    movel([0.119613, -1.324282, -2.607686, -0.780421, 1.570796, 1.690410],accel_mss,speed_ms,0,blend_radius_m)
    movel([0.119842, -1.324467, -2.607569, -0.780352, 1.570796, 1.690638],accel_mss,speed_ms,0,blend_radius_m)
    movel([0.121399, -1.324125, -2.607784, -0.780480, 1.570796, 1.692195],accel_mss,speed_ms,0,blend_radius_m)
    movel([0.123082, -1.323676, -2.608066, -0.780647, 1.570796, 1.693878],accel_mss,speed_ms,0,blend_radius_m)
    movel([0.126728, -1.322614, -2.608731, -0.781044, 1.570796, 1.697525],accel_mss,speed_ms,0,blend_radius_m)
    movel([0.135559, -1.320026, -2.610347, -0.782016, 1.570796, 1.706355],accel_mss,speed_ms,0,blend_radius_m)
    movel([0.136875, -1.312057, -2.615265, -0.785067, 1.570796, 1.707671],accel_mss,speed_ms,0,blend_radius_m)
    movel([0.137268, -1.309610, -2.616758, -0.786021, 1.570796, 1.708065],accel_mss,speed_ms,0,blend_radius_m)
    movel([0.137372, -1.308887, -2.617198, -0.786304, 1.570796, 1.708168],accel_mss,speed_ms,0,blend_radius_m)
    movel([0.137487, -1.307784, -2.617868, -0.786738, 1.570796, 1.708283],accel_mss,speed_ms,0,blend_radius_m)
    movel([0.137501, -1.307407, -2.618096, -0.786886, 1.570796, 1.708297],accel_mss,speed_ms,0,blend_radius_m)
    movel([0.137496, -1.307037, -2.618320, -0.787032, 1.570796, 1.708292],accel_mss,speed_ms,0,blend_radius_m)
    movel([0.137349, -1.306827, -2.618447, -0.787115, 1.570796, 1.708145],accel_mss,speed_ms,0,blend_radius_m)
    movel([0.137251, -1.309745, -2.619823, -0.782821, 1.570796, 1.708047],accel_mss,speed_ms,0,blend_radius_m)
    movel([0.136956, -1.309738, -2.619827, -0.782824, 1.570796, 1.707752],accel_mss,speed_ms,0,blend_radius_m)
    movel([0.136646, -1.309759, -2.619814, -0.782816, 1.570796, 1.707442],accel_mss,speed_ms,0,blend_radius_m)
    movel([0.136330, -1.309805, -2.619786, -0.782797, 1.570796, 1.707126],accel_mss,speed_ms,0,blend_radius_m)
    movel([0.136004, -1.309880, -2.619741, -0.782768, 1.570796, 1.706800],accel_mss,speed_ms,0,blend_radius_m)
    movel([0.130263, -1.311569, -2.618712, -0.782108, 1.570796, 1.701060],accel_mss,speed_ms,0,blend_radius_m)
    movel([0.122240, -1.314022, -2.617212, -0.781155, 1.570796, 1.693036],accel_mss,speed_ms,0,blend_radius_m)
    movel([0.121881, -1.314196, -2.617105, -0.781088, 1.570796, 1.692677],accel_mss,speed_ms,0,blend_radius_m)
    movel([0.121557, -1.314459, -2.616944, -0.780986, 1.570796, 1.692353],accel_mss,speed_ms,0,blend_radius_m)
    movel([0.121274, -1.314831, -2.616715, -0.780843, 1.570796, 1.692071],accel_mss,speed_ms,0,blend_radius_m)
    movel([0.121125, -1.315219, -2.616477, -0.780693, 1.570796, 1.691922],accel_mss,speed_ms,0,blend_radius_m)
    movel([0.120597, -1.318726, -2.614312, -0.779350, 1.570796, 1.691393],accel_mss,speed_ms,0,blend_radius_m)
    movel([0.120081, -1.322273, -2.612107, -0.778009, 1.570796, 1.690877],accel_mss,speed_ms,0,blend_radius_m)
    movel([0.119488, -1.326560, -2.609418, -0.776411, 1.570796, 1.690285],accel_mss,speed_ms,0,blend_radius_m)
    movel([0.119491, -1.326786, -2.609276, -0.776327, 1.570796, 1.690287],accel_mss,speed_ms,0,blend_radius_m)
    movel([0.119613, -1.327186, -2.609024, -0.776179, 1.570796, 1.690410],accel_mss,speed_ms,0,blend_radius_m)
    movel([0.119842, -1.327371, -2.608907, -0.776111, 1.570796, 1.690638],accel_mss,speed_ms,0,blend_radius_m)
    movel([0.121399, -1.327030, -2.609122, -0.776237, 1.570796, 1.692195],accel_mss,speed_ms,0,blend_radius_m)
    movel([0.123082, -1.326582, -2.609405, -0.776403, 1.570796, 1.693878],accel_mss,speed_ms,0,blend_radius_m)
    movel([0.126728, -1.325522, -2.610072, -0.776796, 1.570796, 1.697525],accel_mss,speed_ms,0,blend_radius_m)
    movel([0.135559, -1.322939, -2.611691, -0.777759, 1.570796, 1.706355],accel_mss,speed_ms,0,blend_radius_m)
    movel([0.136875, -1.314985, -2.616621, -0.780783, 1.570796, 1.707671],accel_mss,speed_ms,0,blend_radius_m)
    movel([0.137268, -1.312544, -2.618117, -0.781728, 1.570796, 1.708065],accel_mss,speed_ms,0,blend_radius_m)
    movel([0.137372, -1.311822, -2.618558, -0.782009, 1.570796, 1.708168],accel_mss,speed_ms,0,blend_radius_m)
    movel([0.137487, -1.310721, -2.619229, -0.782439, 1.570796, 1.708283],accel_mss,speed_ms,0,blend_radius_m)
    movel([0.137501, -1.310344, -2.619458, -0.782586, 1.570796, 1.708297],accel_mss,speed_ms,0,blend_radius_m)
    movel([0.137496, -1.309975, -2.619683, -0.782731, 1.570796, 1.708292],accel_mss,speed_ms,0,blend_radius_m)
    movel([0.137349, -1.309765, -2.619810, -0.782813, 1.570796, 1.708145],accel_mss,speed_ms,0,blend_radius_m)
    movel([0.137251, -1.275756, -2.603080, -0.833553, 1.570796, 1.708047],accel_mss,speed_ms,0,blend_radius_m)
    speed_ms = 1.000
    movel([0.134220, -1.265196, -2.609125, -0.838068, 1.570796, 1.705016],accel_mss,speed_ms,0,blend_radius_m)
    speed_ms = 0.008
    movel([0.134220, -1.292915, -2.623010, -0.796463, 1.570796, 1.705016],accel_mss,speed_ms,0,blend_radius_m)
    speed_ms = 0.003
    movel([0.134220, -1.296430, -2.624667, -0.791291, 1.570796, 1.705016],accel_mss,speed_ms,0,blend_radius_m)
    speed_ms = 0.008
    movel([0.121435, -1.300332, -2.622350, -0.789708, 1.570796, 1.692232],accel_mss,speed_ms,0,blend_radius_m)
    movel([0.125336, -1.272015, -2.638732, -0.801642, 1.570796, 1.696133],accel_mss,speed_ms,0,blend_radius_m)
    movel([0.151954, -1.263834, -2.643278, -0.805277, 1.570796, 1.722750],accel_mss,speed_ms,0,blend_radius_m)
    movel([0.147041, -1.292633, -2.626904, -0.792852, 1.570796, 1.717838],accel_mss,speed_ms,0,blend_radius_m)
    movel([0.134220, -1.296430, -2.624667, -0.791291, 1.570796, 1.705016],accel_mss,speed_ms,0,blend_radius_m)
    movel([0.134220, -1.299389, -2.626045, -0.786955, 1.570796, 1.705016],accel_mss,speed_ms,0,blend_radius_m)
    movel([0.121435, -1.303283, -2.623722, -0.785384, 1.570796, 1.692232],accel_mss,speed_ms,0,blend_radius_m)
    movel([0.125336, -1.275018, -2.640145, -0.797226, 1.570796, 1.696133],accel_mss,speed_ms,0,blend_radius_m)
    movel([0.151954, -1.266851, -2.644703, -0.800836, 1.570796, 1.722750],accel_mss,speed_ms,0,blend_radius_m)
    movel([0.147041, -1.295599, -2.628288, -0.788502, 1.570796, 1.717838],accel_mss,speed_ms,0,blend_radius_m)
    movel([0.134220, -1.299389, -2.626045, -0.786955, 1.570796, 1.705016],accel_mss,speed_ms,0,blend_radius_m)
    movel([0.134220, -1.265196, -2.609125, -0.838068, 1.570796, 1.705016],accel_mss,speed_ms,0,blend_radius_m)
    speed_ms = 1.000
    movel([0.114823, -1.278281, -2.601614, -0.832493, 1.570796, 1.685620],accel_mss,speed_ms,0,blend_radius_m)
    speed_ms = 0.008
    movel([0.114823, -1.305800, -2.615320, -0.791269, 1.570796, 1.685620],accel_mss,speed_ms,0,blend_radius_m)
    speed_ms = 0.003
    movel([0.114823, -1.309286, -2.616955, -0.786148, 1.570796, 1.685620],accel_mss,speed_ms,0,blend_radius_m)
    speed_ms = 0.008
    movel([0.111494, -1.310224, -2.616384, -0.785781, 1.570796, 1.682291],accel_mss,speed_ms,0,blend_radius_m)
    movel([0.112360, -1.301984, -2.621362, -0.789043, 1.570796, 1.683156],accel_mss,speed_ms,0,blend_radius_m)
    movel([0.119291, -1.299848, -2.622638, -0.789903, 1.570796, 1.690087],accel_mss,speed_ms,0,blend_radius_m)
    movel([0.118154, -1.308355, -2.617521, -0.786513, 1.570796, 1.688951],accel_mss,speed_ms,0,blend_radius_m)
    movel([0.114823, -1.309286, -2.616955, -0.786148, 1.570796, 1.685620],accel_mss,speed_ms,0,blend_radius_m)
    movel([0.114823, -1.312220, -2.618315, -0.781854, 1.570796, 1.685620],accel_mss,speed_ms,0,blend_radius_m)
    movel([0.111494, -1.313156, -2.617742, -0.781490, 1.570796, 1.682291],accel_mss,speed_ms,0,blend_radius_m)
    movel([0.112360, -1.304932, -2.622732, -0.784725, 1.570796, 1.683156],accel_mss,speed_ms,0,blend_radius_m)
    movel([0.119291, -1.302800, -2.624011, -0.785578, 1.570796, 1.690087],accel_mss,speed_ms,0,blend_radius_m)
    movel([0.118154, -1.311291, -2.618882, -0.782216, 1.570796, 1.688951],accel_mss,speed_ms,0,blend_radius_m)
    movel([0.114823, -1.312220, -2.618315, -0.781854, 1.570796, 1.685620],accel_mss,speed_ms,0,blend_radius_m)
    movel([0.114823, -1.278281, -2.601614, -0.832493, 1.570796, 1.685620],accel_mss,speed_ms,0,blend_radius_m)
    speed_ms = 1.000
    movel([0.107172, -1.280673, -2.600219, -0.831497, 1.570796, 1.677968],accel_mss,speed_ms,0,blend_radius_m)
    speed_ms = 0.008
    movel([0.107172, -1.308154, -2.613892, -0.790343, 1.570796, 1.677968],accel_mss,speed_ms,0,blend_radius_m)
    speed_ms = 0.003
    movel([0.107172, -1.311635, -2.615523, -0.785231, 1.570796, 1.677968],accel_mss,speed_ms,0,blend_radius_m)
    speed_ms = 0.008
    movel([0.103829, -1.312752, -2.614840, -0.784798, 1.570796, 1.674626],accel_mss,speed_ms,0,blend_radius_m)
    movel([0.104823, -1.304343, -2.619946, -0.788100, 1.570796, 1.675619],accel_mss,speed_ms,0,blend_radius_m)
    movel([0.108440, -1.303209, -2.620628, -0.788553, 1.570796, 1.679236],accel_mss,speed_ms,0,blend_radius_m)
    movel([0.109972, -1.302762, -2.620896, -0.788731, 1.570796, 1.680768],accel_mss,speed_ms,0,blend_radius_m)
    movel([0.111330, -1.302426, -2.621097, -0.788866, 1.570796, 1.682127],accel_mss,speed_ms,0,blend_radius_m)
    movel([0.111543, -1.302531, -2.621035, -0.788824, 1.570796, 1.682340],accel_mss,speed_ms,0,blend_radius_m)
    movel([0.111448, -1.303792, -2.620278, -0.788320, 1.570796, 1.682244],accel_mss,speed_ms,0,blend_radius_m)
    movel([0.111288, -1.305189, -2.619436, -0.787763, 1.570796, 1.682084],accel_mss,speed_ms,0,blend_radius_m)
    movel([0.111124, -1.306390, -2.618711, -0.787288, 1.570796, 1.681920],accel_mss,speed_ms,0,blend_radius_m)
    movel([0.110517, -1.310524, -2.616201, -0.785664, 1.570796, 1.681314],accel_mss,speed_ms,0,blend_radius_m)
    movel([0.107172, -1.311635, -2.615523, -0.785231, 1.570796, 1.677968],accel_mss,speed_ms,0,blend_radius_m)
    movel([0.107172, -1.314564, -2.616879, -0.780946, 1.570796, 1.677968],accel_mss,speed_ms,0,blend_radius_m)
    movel([0.103829, -1.315679, -2.616194, -0.780516, 1.570796, 1.674626],accel_mss,speed_ms,0,blend_radius_m)
    movel([0.104823, -1.307287, -2.621312, -0.783790, 1.570796, 1.675619],accel_mss,speed_ms,0,blend_radius_m)
    movel([0.108440, -1.306154, -2.621996, -0.784238, 1.570796, 1.679236],accel_mss,speed_ms,0,blend_radius_m)
    movel([0.109972, -1.305709, -2.622264, -0.784415, 1.570796, 1.680768],accel_mss,speed_ms,0,blend_radius_m)
    movel([0.111330, -1.305373, -2.622467, -0.784549, 1.570796, 1.682127],accel_mss,speed_ms,0,blend_radius_m)
    movel([0.111543, -1.305478, -2.622404, -0.784507, 1.570796, 1.682340],accel_mss,speed_ms,0,blend_radius_m)
    movel([0.111448, -1.306736, -2.621645, -0.784008, 1.570796, 1.682244],accel_mss,speed_ms,0,blend_radius_m)
    movel([0.111288, -1.308132, -2.620801, -0.783456, 1.570796, 1.682084],accel_mss,speed_ms,0,blend_radius_m)
    movel([0.111124, -1.309330, -2.620075, -0.782984, 1.570796, 1.681920],accel_mss,speed_ms,0,blend_radius_m)
    movel([0.110517, -1.313456, -2.617559, -0.781374, 1.570796, 1.681314],accel_mss,speed_ms,0,blend_radius_m)
    movel([0.107172, -1.314564, -2.616879, -0.780946, 1.570796, 1.677968],accel_mss,speed_ms,0,blend_radius_m)
    movel([0.107172, -1.280673, -2.600219, -0.831497, 1.570796, 1.677968],accel_mss,speed_ms,0,blend_radius_m)
    speed_ms = 1.000
    movel([0.109893, -1.289715, -2.594880, -0.827794, 1.570796, 1.680690],accel_mss,speed_ms,0,blend_radius_m)
    speed_ms = 0.008
    movel([0.109893, -1.317050, -2.608430, -0.786910, 1.570796, 1.680690],accel_mss,speed_ms,0,blend_radius_m)
    speed_ms = 0.003
    movel([0.109893, -1.320510, -2.610045, -0.781834, 1.570796, 1.680690],accel_mss,speed_ms,0,blend_radius_m)
    speed_ms = 0.008
    movel([0.102339, -1.322814, -2.608606, -0.780969, 1.570796, 1.673135],accel_mss,speed_ms,0,blend_radius_m)
    movel([0.103372, -1.313982, -2.614084, -0.784322, 1.570796, 1.674168],accel_mss,speed_ms,0,blend_radius_m)
    movel([0.118654, -1.309301, -2.616946, -0.786142, 1.570796, 1.689450],accel_mss,speed_ms,0,blend_radius_m)
    movel([0.117462, -1.318241, -2.611456, -0.782692, 1.570796, 1.688259],accel_mss,speed_ms,0,blend_radius_m)
    movel([0.109893, -1.320510, -2.610045, -0.781834, 1.570796, 1.680690],accel_mss,speed_ms,0,blend_radius_m)
    movel([0.109893, -1.323422, -2.611389, -0.777578, 1.570796, 1.680690],accel_mss,speed_ms,0,blend_radius_m)
    movel([0.102339, -1.325721, -2.609947, -0.776722, 1.570796, 1.673135],accel_mss,speed_ms,0,blend_radius_m)
    movel([0.103372, -1.316907, -2.615437, -0.780045, 1.570796, 1.674168],accel_mss,speed_ms,0,blend_radius_m)
    movel([0.118654, -1.312235, -2.618305, -0.781848, 1.570796, 1.689450],accel_mss,speed_ms,0,blend_radius_m)
    movel([0.117462, -1.321157, -2.612802, -0.778429, 1.570796, 1.688259],accel_mss,speed_ms,0,blend_radius_m)
    movel([0.109893, -1.323422, -2.611389, -0.777578, 1.570796, 1.680690],accel_mss,speed_ms,0,blend_radius_m)
    movel([0.109893, -1.289715, -2.594880, -0.827794, 1.570796, 1.680690],accel_mss,speed_ms,0,blend_radius_m)
    speed_ms = 1.000
    movel([0.109485, -1.291792, -2.593639, -0.826958, 1.570796, 1.680281],accel_mss,speed_ms,0,blend_radius_m)
    speed_ms = 0.008
    movel([0.109485, -1.319092, -2.607160, -0.786136, 1.570796, 1.680281],accel_mss,speed_ms,0,blend_radius_m)
    speed_ms = 0.003
    movel([0.109485, -1.322548, -2.608773, -0.781068, 1.570796, 1.680281],accel_mss,speed_ms,0,blend_radius_m)
    speed_ms = 0.008
    movel([0.104783, -1.323962, -2.607886, -0.780540, 1.570796, 1.675580],accel_mss,speed_ms,0,blend_radius_m)
    movel([0.104081, -1.324156, -2.607765, -0.780468, 1.570796, 1.674877],accel_mss,speed_ms,0,blend_radius_m)
    movel([0.103386, -1.324325, -2.607658, -0.780405, 1.570796, 1.674182],accel_mss,speed_ms,0,blend_radius_m)
    movel([0.102993, -1.324382, -2.607623, -0.780384, 1.570796, 1.673789],accel_mss,speed_ms,0,blend_radius_m)
    movel([0.102649, -1.324372, -2.607629, -0.780388, 1.570796, 1.673445],accel_mss,speed_ms,0,blend_radius_m)
    movel([0.102493, -1.324190, -2.607743, -0.780455, 1.570796, 1.673289],accel_mss,speed_ms,0,blend_radius_m)
    movel([0.102588, -1.323905, -2.607922, -0.780562, 1.570796, 1.673384],accel_mss,speed_ms,0,blend_radius_m)
    movel([0.102959, -1.323614, -2.608105, -0.780670, 1.570796, 1.673756],accel_mss,speed_ms,0,blend_radius_m)
    movel([0.103382, -1.323398, -2.608240, -0.780751, 1.570796, 1.674178],accel_mss,speed_ms,0,blend_radius_m)
    movel([0.104277, -1.323067, -2.608448, -0.780874, 1.570796, 1.675073],accel_mss,speed_ms,0,blend_radius_m)
    movel([0.104940, -1.322847, -2.608586, -0.780957, 1.570796, 1.675736],accel_mss,speed_ms,0,blend_radius_m)
    movel([0.109626, -1.321412, -2.609483, -0.781494, 1.570796, 1.680422],accel_mss,speed_ms,0,blend_radius_m)
    movel([0.114312, -1.320015, -2.610354, -0.782020, 1.570796, 1.685109],accel_mss,speed_ms,0,blend_radius_m)
    movel([0.114972, -1.319836, -2.610465, -0.782088, 1.570796, 1.685769],accel_mss,speed_ms,0,blend_radius_m)
    movel([0.115630, -1.319677, -2.610564, -0.782148, 1.570796, 1.686426],accel_mss,speed_ms,0,blend_radius_m)
    movel([0.116057, -1.319605, -2.610609, -0.782175, 1.570796, 1.686853],accel_mss,speed_ms,0,blend_radius_m)
    movel([0.116443, -1.319609, -2.610606, -0.782174, 1.570796, 1.687239],accel_mss,speed_ms,0,blend_radius_m)
    movel([0.116618, -1.319746, -2.610521, -0.782122, 1.570796, 1.687415],accel_mss,speed_ms,0,blend_radius_m)
    movel([0.116565, -1.320034, -2.610341, -0.782013, 1.570796, 1.687361],accel_mss,speed_ms,0,blend_radius_m)
    movel([0.116232, -1.320332, -2.610156, -0.781901, 1.570796, 1.687028],accel_mss,speed_ms,0,blend_radius_m)
    movel([0.115817, -1.320552, -2.610019, -0.781818, 1.570796, 1.686613],accel_mss,speed_ms,0,blend_radius_m)
    movel([0.114902, -1.320892, -2.609807, -0.781690, 1.570796, 1.685698],accel_mss,speed_ms,0,blend_radius_m)
    movel([0.114192, -1.321124, -2.609662, -0.781602, 1.570796, 1.684988],accel_mss,speed_ms,0,blend_radius_m)
    movel([0.109485, -1.322548, -2.608773, -0.781068, 1.570796, 1.680281],accel_mss,speed_ms,0,blend_radius_m)
    movel([0.109485, -1.325456, -2.610113, -0.776820, 1.570796, 1.680281],accel_mss,speed_ms,0,blend_radius_m)
    movel([0.104783, -1.326867, -2.609225, -0.776297, 1.570796, 1.675580],accel_mss,speed_ms,0,blend_radius_m)
    movel([0.104081, -1.327061, -2.609103, -0.776226, 1.570796, 1.674877],accel_mss,speed_ms,0,blend_radius_m)
    movel([0.103386, -1.327229, -2.608996, -0.776163, 1.570796, 1.674182],accel_mss,speed_ms,0,blend_radius_m)
    movel([0.102993, -1.327286, -2.608961, -0.776142, 1.570796, 1.673789],accel_mss,speed_ms,0,blend_radius_m)
    movel([0.102649, -1.327276, -2.608967, -0.776146, 1.570796, 1.673445],accel_mss,speed_ms,0,blend_radius_m)
    movel([0.102493, -1.327095, -2.609081, -0.776213, 1.570796, 1.673289],accel_mss,speed_ms,0,blend_radius_m)
    movel([0.102588, -1.326810, -2.609261, -0.776318, 1.570796, 1.673384],accel_mss,speed_ms,0,blend_radius_m)
    movel([0.102959, -1.326519, -2.609444, -0.776426, 1.570796, 1.673756],accel_mss,speed_ms,0,blend_radius_m)
    movel([0.103382, -1.326304, -2.609580, -0.776505, 1.570796, 1.674178],accel_mss,speed_ms,0,blend_radius_m)
    movel([0.104277, -1.325974, -2.609787, -0.776628, 1.570796, 1.675073],accel_mss,speed_ms,0,blend_radius_m)
    movel([0.104940, -1.325754, -2.609926, -0.776709, 1.570796, 1.675736],accel_mss,speed_ms,0,blend_radius_m)
    movel([0.109626, -1.324322, -2.610825, -0.777242, 1.570796, 1.680422],accel_mss,speed_ms,0,blend_radius_m)
    movel([0.114312, -1.322928, -2.611698, -0.777763, 1.570796, 1.685109],accel_mss,speed_ms,0,blend_radius_m)
    movel([0.114972, -1.322750, -2.611809, -0.777830, 1.570796, 1.685769],accel_mss,speed_ms,0,blend_radius_m)
    movel([0.115630, -1.322590, -2.611909, -0.777890, 1.570796, 1.686426],accel_mss,speed_ms,0,blend_radius_m)
    movel([0.116057, -1.322518, -2.611954, -0.777917, 1.570796, 1.686853],accel_mss,speed_ms,0,blend_radius_m)
    movel([0.116443, -1.322522, -2.611951, -0.777916, 1.570796, 1.687239],accel_mss,speed_ms,0,blend_radius_m)
    movel([0.116618, -1.322660, -2.611865, -0.777864, 1.570796, 1.687415],accel_mss,speed_ms,0,blend_radius_m)
    movel([0.116565, -1.322947, -2.611686, -0.777756, 1.570796, 1.687361],accel_mss,speed_ms,0,blend_radius_m)
    movel([0.116232, -1.323244, -2.611500, -0.777645, 1.570796, 1.687028],accel_mss,speed_ms,0,blend_radius_m)
    movel([0.115817, -1.323463, -2.611363, -0.777563, 1.570796, 1.686613],accel_mss,speed_ms,0,blend_radius_m)
    movel([0.114902, -1.323803, -2.611150, -0.777436, 1.570796, 1.685698],accel_mss,speed_ms,0,blend_radius_m)
    movel([0.114192, -1.324035, -2.611005, -0.777349, 1.570796, 1.684988],accel_mss,speed_ms,0,blend_radius_m)
    movel([0.109485, -1.325456, -2.610113, -0.776820, 1.570796, 1.680281],accel_mss,speed_ms,0,blend_radius_m)
    movel([0.109485, -1.291792, -2.593639, -0.826958, 1.570796, 1.680281],accel_mss,speed_ms,0,blend_radius_m)
    speed_ms = 1.000
    movel([0.109344, -1.292948, -2.592946, -0.826495, 1.570796, 1.680140],accel_mss,speed_ms,0,blend_radius_m)
    speed_ms = 0.008
    movel([0.109344, -1.320229, -2.606452, -0.785708, 1.570796, 1.680140],accel_mss,speed_ms,0,blend_radius_m)
    speed_ms = 0.003
    movel([0.109344, -1.323682, -2.608062, -0.780645, 1.570796, 1.680140],accel_mss,speed_ms,0,blend_radius_m)
    speed_ms = 0.008
    movel([0.106080, -1.324648, -2.607456, -0.780285, 1.570796, 1.676877],accel_mss,speed_ms,0,blend_radius_m)
    movel([0.104022, -1.325217, -2.607098, -0.780074, 1.570796, 1.674818],accel_mss,speed_ms,0,blend_radius_m)
    movel([0.102440, -1.325630, -2.606838, -0.779921, 1.570796, 1.673237],accel_mss,speed_ms,0,blend_radius_m)
    movel([0.102423, -1.325400, -2.606983, -0.780007, 1.570796, 1.673220],accel_mss,speed_ms,0,blend_radius_m)
    movel([0.104260, -1.324746, -2.607394, -0.780249, 1.570796, 1.675057],accel_mss,speed_ms,0,blend_radius_m)
    movel([0.106216, -1.324101, -2.607799, -0.780489, 1.570796, 1.677012],accel_mss,speed_ms,0,blend_radius_m)
    movel([0.109414, -1.323115, -2.608418, -0.780856, 1.570796, 1.680211],accel_mss,speed_ms,0,blend_radius_m)
    movel([0.112608, -1.322175, -2.609006, -0.781208, 1.570796, 1.683404],accel_mss,speed_ms,0,blend_radius_m)
    movel([0.114555, -1.321644, -2.609338, -0.781407, 1.570796, 1.685351],accel_mss,speed_ms,0,blend_radius_m)
    movel([0.116327, -1.321197, -2.609617, -0.781575, 1.570796, 1.687123],accel_mss,speed_ms,0,blend_radius_m)
    movel([0.116348, -1.321426, -2.609474, -0.781489, 1.570796, 1.687144],accel_mss,speed_ms,0,blend_radius_m)
    movel([0.114690, -1.322005, -2.609113, -0.781272, 1.570796, 1.685487],accel_mss,speed_ms,0,blend_radius_m)
    movel([0.112613, -1.322681, -2.608689, -0.781018, 1.570796, 1.683409],accel_mss,speed_ms,0,blend_radius_m)
    movel([0.109344, -1.323682, -2.608062, -0.780645, 1.570796, 1.680140],accel_mss,speed_ms,0,blend_radius_m)
    movel([0.109344, -1.326588, -2.609401, -0.776400, 1.570796, 1.680140],accel_mss,speed_ms,0,blend_radius_m)
    movel([0.106080, -1.327551, -2.608793, -0.776044, 1.570796, 1.676877],accel_mss,speed_ms,0,blend_radius_m)
    movel([0.104022, -1.328120, -2.608434, -0.775835, 1.570796, 1.674818],accel_mss,speed_ms,0,blend_radius_m)
    movel([0.102440, -1.328531, -2.608174, -0.775684, 1.570796, 1.673237],accel_mss,speed_ms,0,blend_radius_m)
    movel([0.102423, -1.328301, -2.608319, -0.775768, 1.570796, 1.673220],accel_mss,speed_ms,0,blend_radius_m)
    movel([0.104260, -1.327649, -2.608732, -0.776008, 1.570796, 1.675057],accel_mss,speed_ms,0,blend_radius_m)
    movel([0.106216, -1.327005, -2.609138, -0.776246, 1.570796, 1.677012],accel_mss,speed_ms,0,blend_radius_m)
    movel([0.109414, -1.326022, -2.609757, -0.776610, 1.570796, 1.680211],accel_mss,speed_ms,0,blend_radius_m)
    movel([0.112608, -1.325083, -2.610347, -0.776959, 1.570796, 1.683404],accel_mss,speed_ms,0,blend_radius_m)
    movel([0.114555, -1.324553, -2.610680, -0.777156, 1.570796, 1.685351],accel_mss,speed_ms,0,blend_radius_m)
    movel([0.116327, -1.324108, -2.610959, -0.777322, 1.570796, 1.687123],accel_mss,speed_ms,0,blend_radius_m)
    movel([0.116348, -1.324336, -2.610816, -0.777237, 1.570796, 1.687144],accel_mss,speed_ms,0,blend_radius_m)
    movel([0.114690, -1.324913, -2.610454, -0.777022, 1.570796, 1.685487],accel_mss,speed_ms,0,blend_radius_m)
    movel([0.112613, -1.325589, -2.610030, -0.776771, 1.570796, 1.683409],accel_mss,speed_ms,0,blend_radius_m)
    movel([0.109344, -1.326588, -2.609401, -0.776400, 1.570796, 1.680140],accel_mss,speed_ms,0,blend_radius_m)
    movel([0.109344, -1.292948, -2.592946, -0.826495, 1.570796, 1.680140],accel_mss,speed_ms,0,blend_radius_m)
    speed_ms = 1.000
    movel([0.109203, -1.294102, -2.592252, -0.826034, 1.570796, 1.680000],accel_mss,speed_ms,0,blend_radius_m)
    speed_ms = 0.008
    movel([0.109203, -1.321364, -2.605743, -0.785282, 1.570796, 1.680000],accel_mss,speed_ms,0,blend_radius_m)
    speed_ms = 0.003
    movel([0.109203, -1.324814, -2.607351, -0.780224, 1.570796, 1.680000],accel_mss,speed_ms,0,blend_radius_m)
    speed_ms = 0.008
    movel([0.105944, -1.325777, -2.606745, -0.779867, 1.570796, 1.676740],accel_mss,speed_ms,0,blend_radius_m)
    movel([0.103888, -1.326345, -2.606387, -0.779657, 1.570796, 1.674685],accel_mss,speed_ms,0,blend_radius_m)
    movel([0.102309, -1.326756, -2.606127, -0.779505, 1.570796, 1.673105],accel_mss,speed_ms,0,blend_radius_m)
    movel([0.102292, -1.326526, -2.606273, -0.779590, 1.570796, 1.673088],accel_mss,speed_ms,0,blend_radius_m)
    movel([0.104126, -1.325874, -2.606684, -0.779831, 1.570796, 1.674923],accel_mss,speed_ms,0,blend_radius_m)
    movel([0.106079, -1.325231, -2.607089, -0.780069, 1.570796, 1.676876],accel_mss,speed_ms,0,blend_radius_m)
    movel([0.109274, -1.324248, -2.607707, -0.780434, 1.570796, 1.680070],accel_mss,speed_ms,0,blend_radius_m)
    movel([0.112463, -1.323311, -2.608295, -0.780783, 1.570796, 1.683259],accel_mss,speed_ms,0,blend_radius_m)
    movel([0.114407, -1.322781, -2.608627, -0.780981, 1.570796, 1.685203],accel_mss,speed_ms,0,blend_radius_m)
    movel([0.116177, -1.322336, -2.608905, -0.781148, 1.570796, 1.686973],accel_mss,speed_ms,0,blend_radius_m)
    movel([0.116198, -1.322564, -2.608762, -0.781062, 1.570796, 1.686994],accel_mss,speed_ms,0,blend_radius_m)
    movel([0.114543, -1.323142, -2.608401, -0.780846, 1.570796, 1.685339],accel_mss,speed_ms,0,blend_radius_m)
    movel([0.112468, -1.323816, -2.607978, -0.780595, 1.570796, 1.683264],accel_mss,speed_ms,0,blend_radius_m)
    movel([0.109203, -1.324814, -2.607351, -0.780224, 1.570796, 1.680000],accel_mss,speed_ms,0,blend_radius_m)
    movel([0.109203, -1.327717, -2.608688, -0.775983, 1.570796, 1.680000],accel_mss,speed_ms,0,blend_radius_m)
    movel([0.105944, -1.328678, -2.608081, -0.775630, 1.570796, 1.676740],accel_mss,speed_ms,0,blend_radius_m)
    movel([0.103888, -1.329245, -2.607722, -0.775422, 1.570796, 1.674685],accel_mss,speed_ms,0,blend_radius_m)
    movel([0.102309, -1.329655, -2.607462, -0.775272, 1.570796, 1.673105],accel_mss,speed_ms,0,blend_radius_m)
    movel([0.102292, -1.329426, -2.607607, -0.775356, 1.570796, 1.673088],accel_mss,speed_ms,0,blend_radius_m)
    movel([0.104126, -1.328775, -2.608020, -0.775594, 1.570796, 1.674923],accel_mss,speed_ms,0,blend_radius_m)
    movel([0.106079, -1.328133, -2.608426, -0.775830, 1.570796, 1.676876],accel_mss,speed_ms,0,blend_radius_m)
    movel([0.109274, -1.327153, -2.609045, -0.776192, 1.570796, 1.680070],accel_mss,speed_ms,0,blend_radius_m)
    movel([0.112463, -1.326217, -2.609635, -0.776538, 1.570796, 1.683259],accel_mss,speed_ms,0,blend_radius_m)
    movel([0.114407, -1.325689, -2.609967, -0.776734, 1.570796, 1.685203],accel_mss,speed_ms,0,blend_radius_m)
    movel([0.116177, -1.325244, -2.610246, -0.776899, 1.570796, 1.686973],accel_mss,speed_ms,0,blend_radius_m)
    movel([0.116198, -1.325472, -2.610103, -0.776814, 1.570796, 1.686994],accel_mss,speed_ms,0,blend_radius_m)
    movel([0.114543, -1.326048, -2.609741, -0.776600, 1.570796, 1.685339],accel_mss,speed_ms,0,blend_radius_m)
    movel([0.112468, -1.326721, -2.609317, -0.776351, 1.570796, 1.683264],accel_mss,speed_ms,0,blend_radius_m)
    movel([0.109203, -1.327717, -2.608688, -0.775983, 1.570796, 1.680000],accel_mss,speed_ms,0,blend_radius_m)
    movel([0.109203, -1.294102, -2.592252, -0.826034, 1.570796, 1.680000],accel_mss,speed_ms,0,blend_radius_m)
    speed_ms = 1.000
    movel([0.112615, -1.314973, -2.579420, -0.817996, 1.570796, 1.683412],accel_mss,speed_ms,0,blend_radius_m)
    speed_ms = 0.008
    movel([0.112615, -1.341877, -2.592627, -0.777885, 1.570796, 1.683412],accel_mss,speed_ms,0,blend_radius_m)
    speed_ms = 0.003
    movel([0.112615, -1.345277, -2.594201, -0.772911, 1.570796, 1.683412],accel_mss,speed_ms,0,blend_radius_m)
    speed_ms = 0.008
    movel([0.111947, -1.345445, -2.594091, -0.772854, 1.570796, 1.682743],accel_mss,speed_ms,0,blend_radius_m)
    movel([0.108003, -1.346284, -2.593539, -0.772566, 1.570796, 1.678799],accel_mss,speed_ms,0,blend_radius_m)
    movel([0.101292, -1.347670, -2.592625, -0.772094, 1.570796, 1.672089],accel_mss,speed_ms,0,blend_radius_m)
    movel([0.099538, -1.348042, -2.592380, -0.771967, 1.570796, 1.670334],accel_mss,speed_ms,0,blend_radius_m)
    movel([0.099271, -1.348071, -2.592361, -0.771957, 1.570796, 1.670067],accel_mss,speed_ms,0,blend_radius_m)
    movel([0.099589, -1.344674, -2.594596, -0.773119, 1.570796, 1.670385],accel_mss,speed_ms,0,blend_radius_m)
    movel([0.099930, -1.341512, -2.596663, -0.774214, 1.570796, 1.670726],accel_mss,speed_ms,0,blend_radius_m)
    movel([0.100273, -1.338611, -2.598547, -0.775231, 1.570796, 1.671069],accel_mss,speed_ms,0,blend_radius_m)
    movel([0.101573, -1.328076, -2.605293, -0.779020, 1.570796, 1.672369],accel_mss,speed_ms,0,blend_radius_m)
    movel([0.116462, -1.323461, -2.608201, -0.780727, 1.570796, 1.687259],accel_mss,speed_ms,0,blend_radius_m)
    movel([0.113646, -1.344982, -2.594394, -0.773013, 1.570796, 1.684442],accel_mss,speed_ms,0,blend_radius_m)
    movel([0.112615, -1.345277, -2.594201, -0.772911, 1.570796, 1.683412],accel_mss,speed_ms,0,blend_radius_m)
    movel([0.112615, -1.348137, -2.595509, -0.768743, 1.570796, 1.683412],accel_mss,speed_ms,0,blend_radius_m)
    movel([0.111947, -1.348305, -2.595399, -0.768686, 1.570796, 1.682743],accel_mss,speed_ms,0,blend_radius_m)
    movel([0.108003, -1.349142, -2.594845, -0.768401, 1.570796, 1.678799],accel_mss,speed_ms,0,blend_radius_m)
    movel([0.101292, -1.350526, -2.593930, -0.767933, 1.570796, 1.672089],accel_mss,speed_ms,0,blend_radius_m)
    movel([0.099538, -1.350897, -2.593684, -0.767808, 1.570796, 1.670334],accel_mss,speed_ms,0,blend_radius_m)
    movel([0.099271, -1.350925, -2.593665, -0.767799, 1.570796, 1.670067],accel_mss,speed_ms,0,blend_radius_m)
    movel([0.099589, -1.347536, -2.595905, -0.768948, 1.570796, 1.670385],accel_mss,speed_ms,0,blend_radius_m)
    movel([0.099930, -1.344380, -2.597977, -0.770032, 1.570796, 1.670726],accel_mss,speed_ms,0,blend_radius_m)
    movel([0.100273, -1.341485, -2.599865, -0.771039, 1.570796, 1.671069],accel_mss,speed_ms,0,blend_radius_m)
    movel([0.101573, -1.330973, -2.606625, -0.774791, 1.570796, 1.672369],accel_mss,speed_ms,0,blend_radius_m)
    movel([0.116462, -1.326366, -2.609540, -0.776482, 1.570796, 1.687259],accel_mss,speed_ms,0,blend_radius_m)
    movel([0.113646, -1.347843, -2.595703, -0.768843, 1.570796, 1.684442],accel_mss,speed_ms,0,blend_radius_m)
    movel([0.112615, -1.348137, -2.595509, -0.768743, 1.570796, 1.683412],accel_mss,speed_ms,0,blend_radius_m)
    movel([0.112615, -1.314973, -2.579420, -0.817996, 1.570796, 1.683412],accel_mss,speed_ms,0,blend_radius_m)
    speed_ms = 1.000
    movel([0.113566, -1.316583, -2.578407, -0.817399, 1.570796, 1.684362],accel_mss,speed_ms,0,blend_radius_m)
    speed_ms = 0.008
    movel([0.113566, -1.343458, -2.591592, -0.777339, 1.570796, 1.684362],accel_mss,speed_ms,0,blend_radius_m)
    speed_ms = 0.003
    movel([0.113566, -1.346854, -2.593163, -0.772371, 1.570796, 1.684362],accel_mss,speed_ms,0,blend_radius_m)
    speed_ms = 0.008
    movel([0.112789, -1.347059, -2.593029, -0.772302, 1.570796, 1.683585],accel_mss,speed_ms,0,blend_radius_m)
    movel([0.112022, -1.347223, -2.592920, -0.772246, 1.570796, 1.682819],accel_mss,speed_ms,0,blend_radius_m)
    movel([0.107031, -1.348176, -2.592291, -0.771922, 1.570796, 1.677827],accel_mss,speed_ms,0,blend_radius_m)
    movel([0.099261, -1.349677, -2.591298, -0.771414, 1.570796, 1.670057],accel_mss,speed_ms,0,blend_radius_m)
    movel([0.099030, -1.349660, -2.591310, -0.771420, 1.570796, 1.669826],accel_mss,speed_ms,0,blend_radius_m)
    movel([0.099078, -1.349416, -2.591471, -0.771502, 1.570796, 1.669874],accel_mss,speed_ms,0,blend_radius_m)
    movel([0.099655, -1.349215, -2.591604, -0.771570, 1.570796, 1.670451],accel_mss,speed_ms,0,blend_radius_m)
    movel([0.100377, -1.349014, -2.591737, -0.771638, 1.570796, 1.671173],accel_mss,speed_ms,0,blend_radius_m)
    movel([0.101596, -1.348721, -2.591931, -0.771737, 1.570796, 1.672393],accel_mss,speed_ms,0,blend_radius_m)
    movel([0.105858, -1.347817, -2.592528, -0.772044, 1.570796, 1.676654],accel_mss,speed_ms,0,blend_radius_m)
    movel([0.114326, -1.346105, -2.593656, -0.772628, 1.570796, 1.685123],accel_mss,speed_ms,0,blend_radius_m)
    movel([0.114368, -1.346362, -2.593487, -0.772540, 1.570796, 1.685164],accel_mss,speed_ms,0,blend_radius_m)
    movel([0.114160, -1.346593, -2.593336, -0.772461, 1.570796, 1.684957],accel_mss,speed_ms,0,blend_radius_m)
    movel([0.113791, -1.346779, -2.593213, -0.772397, 1.570796, 1.684587],accel_mss,speed_ms,0,blend_radius_m)
    movel([0.113566, -1.349711, -2.594469, -0.768208, 1.570796, 1.684362],accel_mss,speed_ms,0,blend_radius_m)
    movel([0.112789, -1.349915, -2.594334, -0.768140, 1.570796, 1.683585],accel_mss,speed_ms,0,blend_radius_m)
    movel([0.112022, -1.350079, -2.594226, -0.768084, 1.570796, 1.682819],accel_mss,speed_ms,0,blend_radius_m)
    movel([0.107031, -1.351030, -2.593595, -0.767763, 1.570796, 1.677827],accel_mss,speed_ms,0,blend_radius_m)
    movel([0.099261, -1.352528, -2.592600, -0.767261, 1.570796, 1.670057],accel_mss,speed_ms,0,blend_radius_m)
    movel([0.099030, -1.352511, -2.592612, -0.767267, 1.570796, 1.669826],accel_mss,speed_ms,0,blend_radius_m)
    movel([0.099078, -1.352267, -2.592773, -0.767348, 1.570796, 1.669874],accel_mss,speed_ms,0,blend_radius_m)
    movel([0.099655, -1.352067, -2.592907, -0.767415, 1.570796, 1.670451],accel_mss,speed_ms,0,blend_radius_m)
    movel([0.100377, -1.351867, -2.593040, -0.767482, 1.570796, 1.671173],accel_mss,speed_ms,0,blend_radius_m)
    movel([0.101596, -1.351574, -2.593235, -0.767581, 1.570796, 1.672393],accel_mss,speed_ms,0,blend_radius_m)
    movel([0.105858, -1.350672, -2.593833, -0.767884, 1.570796, 1.676654],accel_mss,speed_ms,0,blend_radius_m)
    movel([0.114326, -1.348964, -2.594963, -0.768462, 1.570796, 1.685123],accel_mss,speed_ms,0,blend_radius_m)
    movel([0.114368, -1.349220, -2.594794, -0.768375, 1.570796, 1.685164],accel_mss,speed_ms,0,blend_radius_m)
    movel([0.114160, -1.349450, -2.594642, -0.768297, 1.570796, 1.684957],accel_mss,speed_ms,0,blend_radius_m)
    movel([0.113791, -1.349636, -2.594519, -0.768234, 1.570796, 1.684587],accel_mss,speed_ms,0,blend_radius_m)
    movel([0.113566, -1.316583, -2.578407, -0.817399, 1.570796, 1.684362],accel_mss,speed_ms,0,blend_radius_m)
    speed_ms = 1.000
    movel([0.110224, -1.318088, -2.577456, -0.816844, 1.570796, 1.681020],accel_mss,speed_ms,0,blend_radius_m)
    speed_ms = 0.008
    movel([0.110224, -1.344937, -2.590621, -0.776831, 1.570796, 1.681020],accel_mss,speed_ms,0,blend_radius_m)
    speed_ms = 0.003
    movel([0.110224, -1.348329, -2.592190, -0.771870, 1.570796, 1.681020],accel_mss,speed_ms,0,blend_radius_m)
    speed_ms = 0.008
    movel([0.108876, -1.348588, -2.592019, -0.771782, 1.570796, 1.679673],accel_mss,speed_ms,0,blend_radius_m)
    movel([0.107920, -1.348756, -2.591908, -0.771725, 1.570796, 1.678717],accel_mss,speed_ms,0,blend_radius_m)
    movel([0.106683, -1.348952, -2.591778, -0.771659, 1.570796, 1.677480],accel_mss,speed_ms,0,blend_radius_m)
    movel([0.108443, -1.348432, -2.592122, -0.771835, 1.570796, 1.679239],accel_mss,speed_ms,0,blend_radius_m)
    movel([0.109941, -1.348114, -2.592332, -0.771943, 1.570796, 1.680737],accel_mss,speed_ms,0,blend_radius_m)
    movel([0.111339, -1.347838, -2.592514, -0.772036, 1.570796, 1.682135],accel_mss,speed_ms,0,blend_radius_m)
    movel([0.112572, -1.347615, -2.592662, -0.772112, 1.570796, 1.683369],accel_mss,speed_ms,0,blend_radius_m)
    movel([0.114085, -1.347379, -2.592817, -0.772193, 1.570796, 1.684882],accel_mss,speed_ms,0,blend_radius_m)
    movel([0.113798, -1.347551, -2.592704, -0.772134, 1.570796, 1.684594],accel_mss,speed_ms,0,blend_radius_m)
    movel([0.112067, -1.347948, -2.592442, -0.771999, 1.570796, 1.682863],accel_mss,speed_ms,0,blend_radius_m)
    movel([0.110224, -1.348329, -2.592190, -0.771870, 1.570796, 1.681020],accel_mss,speed_ms,0,blend_radius_m)
    movel([0.110224, -1.351183, -2.593494, -0.767712, 1.570796, 1.681020],accel_mss,speed_ms,0,blend_radius_m)
    movel([0.108876, -1.351441, -2.593323, -0.767625, 1.570796, 1.679673],accel_mss,speed_ms,0,blend_radius_m)
    movel([0.107920, -1.351609, -2.593211, -0.767569, 1.570796, 1.678717],accel_mss,speed_ms,0,blend_radius_m)
    movel([0.106683, -1.351805, -2.593081, -0.767503, 1.570796, 1.677480],accel_mss,speed_ms,0,blend_radius_m)
    movel([0.108443, -1.351286, -2.593426, -0.767677, 1.570796, 1.679239],accel_mss,speed_ms,0,blend_radius_m)
    movel([0.109941, -1.350969, -2.593636, -0.767784, 1.570796, 1.680737],accel_mss,speed_ms,0,blend_radius_m)
    movel([0.111339, -1.350693, -2.593819, -0.767877, 1.570796, 1.682135],accel_mss,speed_ms,0,blend_radius_m)
    movel([0.112572, -1.350470, -2.593967, -0.767952, 1.570796, 1.683369],accel_mss,speed_ms,0,blend_radius_m)
    movel([0.114085, -1.350235, -2.594122, -0.768031, 1.570796, 1.684882],accel_mss,speed_ms,0,blend_radius_m)
    movel([0.113798, -1.350407, -2.594009, -0.767974, 1.570796, 1.684594],accel_mss,speed_ms,0,blend_radius_m)
    movel([0.112067, -1.350803, -2.593746, -0.767840, 1.570796, 1.682863],accel_mss,speed_ms,0,blend_radius_m)
    movel([0.110224, -1.351183, -2.593494, -0.767712, 1.570796, 1.681020],accel_mss,speed_ms,0,blend_radius_m)
    movel([0.110224, -1.318088, -2.577456, -0.816844, 1.570796, 1.681020],accel_mss,speed_ms,0,blend_radius_m)
    speed_ms = 1.000
    movel([0.111877, -1.324726, -2.573231, -0.814432, 1.570796, 1.682674],accel_mss,speed_ms,0,blend_radius_m)
    speed_ms = 0.008
    movel([0.111877, -1.351455, -2.586307, -0.774627, 1.570796, 1.682674],accel_mss,speed_ms,0,blend_radius_m)
    speed_ms = 0.003
    movel([0.111877, -1.354831, -2.587864, -0.769694, 1.570796, 1.682674],accel_mss,speed_ms,0,blend_radius_m)
    speed_ms = 0.008
    movel([0.111217, -1.355085, -2.587694, -0.769610, 1.570796, 1.682014],accel_mss,speed_ms,0,blend_radius_m)
    movel([0.110559, -1.355306, -2.587546, -0.769537, 1.570796, 1.681356],accel_mss,speed_ms,0,blend_radius_m)
    movel([0.109957, -1.355481, -2.587428, -0.769479, 1.570796, 1.680753],accel_mss,speed_ms,0,blend_radius_m)
    movel([0.109060, -1.355712, -2.587274, -0.769403, 1.570796, 1.679856],accel_mss,speed_ms,0,blend_radius_m)
    movel([0.108163, -1.355922, -2.587133, -0.769334, 1.570796, 1.678960],accel_mss,speed_ms,0,blend_radius_m)
    movel([0.107268, -1.356106, -2.587009, -0.769274, 1.570796, 1.678064],accel_mss,speed_ms,0,blend_radius_m)
    movel([0.106375, -1.356266, -2.586902, -0.769221, 1.570796, 1.677171],accel_mss,speed_ms,0,blend_radius_m)
    movel([0.105495, -1.356399, -2.586812, -0.769178, 1.570796, 1.676292],accel_mss,speed_ms,0,blend_radius_m)
    movel([0.104906, -1.356473, -2.586763, -0.769154, 1.570796, 1.675702],accel_mss,speed_ms,0,blend_radius_m)
    movel([0.104329, -1.356522, -2.586730, -0.769137, 1.570796, 1.675126],accel_mss,speed_ms,0,blend_radius_m)
    movel([0.103760, -1.356547, -2.586713, -0.769129, 1.570796, 1.674557],accel_mss,speed_ms,0,blend_radius_m)
    movel([0.103212, -1.356547, -2.586713, -0.769129, 1.570796, 1.674008],accel_mss,speed_ms,0,blend_radius_m)
    movel([0.102701, -1.356524, -2.586728, -0.769137, 1.570796, 1.673497],accel_mss,speed_ms,0,blend_radius_m)
    movel([0.102202, -1.356475, -2.586761, -0.769153, 1.570796, 1.672999],accel_mss,speed_ms,0,blend_radius_m)
    movel([0.101717, -1.356402, -2.586810, -0.769177, 1.570796, 1.672513],accel_mss,speed_ms,0,blend_radius_m)
    movel([0.101237, -1.356303, -2.586877, -0.769209, 1.570796, 1.672033],accel_mss,speed_ms,0,blend_radius_m)
    movel([0.100728, -1.356167, -2.586968, -0.769254, 1.570796, 1.671524],accel_mss,speed_ms,0,blend_radius_m)
    movel([0.100237, -1.356004, -2.587077, -0.769307, 1.570796, 1.671034],accel_mss,speed_ms,0,blend_radius_m)
    movel([0.099800, -1.355824, -2.587198, -0.769367, 1.570796, 1.670597],accel_mss,speed_ms,0,blend_radius_m)
    movel([0.099384, -1.355619, -2.587336, -0.769434, 1.570796, 1.670180],accel_mss,speed_ms,0,blend_radius_m)
    movel([0.099020, -1.355400, -2.587483, -0.769506, 1.570796, 1.669817],accel_mss,speed_ms,0,blend_radius_m)
    movel([0.098775, -1.355215, -2.587607, -0.769567, 1.570796, 1.669571],accel_mss,speed_ms,0,blend_radius_m)
    movel([0.098545, -1.354981, -2.587764, -0.769644, 1.570796, 1.669341],accel_mss,speed_ms,0,blend_radius_m)
    movel([0.098351, -1.354719, -2.587939, -0.769731, 1.570796, 1.669147],accel_mss,speed_ms,0,blend_radius_m)
    movel([0.098188, -1.354413, -2.588144, -0.769832, 1.570796, 1.668985],accel_mss,speed_ms,0,blend_radius_m)
    movel([0.098074, -1.354077, -2.588369, -0.769943, 1.570796, 1.668871],accel_mss,speed_ms,0,blend_radius_m)
    movel([0.098004, -1.353702, -2.588619, -0.770067, 1.570796, 1.668801],accel_mss,speed_ms,0,blend_radius_m)
    movel([0.097972, -1.353279, -2.588902, -0.770208, 1.570796, 1.668769],accel_mss,speed_ms,0,blend_radius_m)
    movel([0.097987, -1.352816, -2.589211, -0.770362, 1.570796, 1.668783],accel_mss,speed_ms,0,blend_radius_m)
    movel([0.098044, -1.352378, -2.589503, -0.770508, 1.570796, 1.668840],accel_mss,speed_ms,0,blend_radius_m)
    movel([0.098105, -1.352106, -2.589685, -0.770599, 1.570796, 1.668901],accel_mss,speed_ms,0,blend_radius_m)
    movel([0.098181, -1.351830, -2.589868, -0.770691, 1.570796, 1.668977],accel_mss,speed_ms,0,blend_radius_m)
    movel([0.098380, -1.351486, -2.590097, -0.770806, 1.570796, 1.669176],accel_mss,speed_ms,0,blend_radius_m)
    movel([0.098617, -1.351287, -2.590230, -0.770873, 1.570796, 1.669414],accel_mss,speed_ms,0,blend_radius_m)
    movel([0.098975, -1.351129, -2.590335, -0.770926, 1.570796, 1.669772],accel_mss,speed_ms,0,blend_radius_m)
    movel([0.099661, -1.350970, -2.590440, -0.770979, 1.570796, 1.670458],accel_mss,speed_ms,0,blend_radius_m)
    movel([0.102034, -1.350434, -2.590796, -0.771159, 1.570796, 1.672831],accel_mss,speed_ms,0,blend_radius_m)
    movel([0.104178, -1.349982, -2.591096, -0.771311, 1.570796, 1.674974],accel_mss,speed_ms,0,blend_radius_m)
    movel([0.113737, -1.348117, -2.592330, -0.771942, 1.570796, 1.684533],accel_mss,speed_ms,0,blend_radius_m)
    movel([0.113991, -1.348085, -2.592352, -0.771953, 1.570796, 1.684787],accel_mss,speed_ms,0,blend_radius_m)
    movel([0.113996, -1.348312, -2.592202, -0.771876, 1.570796, 1.684793],accel_mss,speed_ms,0,blend_radius_m)
    movel([0.113949, -1.349169, -2.591634, -0.771585, 1.570796, 1.684746],accel_mss,speed_ms,0,blend_radius_m)
    movel([0.113889, -1.349901, -2.591150, -0.771338, 1.570796, 1.684685],accel_mss,speed_ms,0,blend_radius_m)
    movel([0.113767, -1.350955, -2.590450, -0.770984, 1.570796, 1.684563],accel_mss,speed_ms,0,blend_radius_m)
    movel([0.113343, -1.354235, -2.588263, -0.769891, 1.570796, 1.684139],accel_mss,speed_ms,0,blend_radius_m)
    movel([0.111877, -1.354831, -2.587864, -0.769694, 1.570796, 1.682674],accel_mss,speed_ms,0,blend_radius_m)
    movel([0.111877, -1.357671, -2.589159, -0.765559, 1.570796, 1.682674],accel_mss,speed_ms,0,blend_radius_m)
    movel([0.111217, -1.357924, -2.588989, -0.765476, 1.570796, 1.682014],accel_mss,speed_ms,0,blend_radius_m)
    movel([0.110559, -1.358145, -2.588840, -0.765404, 1.570796, 1.681356],accel_mss,speed_ms,0,blend_radius_m)
    movel([0.109957, -1.358320, -2.588722, -0.765347, 1.570796, 1.680753],accel_mss,speed_ms,0,blend_radius_m)
    movel([0.109060, -1.358550, -2.588567, -0.765272, 1.570796, 1.679856],accel_mss,speed_ms,0,blend_radius_m)
    movel([0.108163, -1.358759, -2.588426, -0.765204, 1.570796, 1.678960],accel_mss,speed_ms,0,blend_radius_m)
    movel([0.107268, -1.358943, -2.588302, -0.765144, 1.570796, 1.678064],accel_mss,speed_ms,0,blend_radius_m)
    movel([0.106375, -1.359102, -2.588194, -0.765092, 1.570796, 1.677171],accel_mss,speed_ms,0,blend_radius_m)
    movel([0.105495, -1.359235, -2.588105, -0.765049, 1.570796, 1.676292],accel_mss,speed_ms,0,blend_radius_m)
    movel([0.104906, -1.359309, -2.588055, -0.765025, 1.570796, 1.675702],accel_mss,speed_ms,0,blend_radius_m)
    movel([0.104329, -1.359358, -2.588022, -0.765009, 1.570796, 1.675126],accel_mss,speed_ms,0,blend_radius_m)
    movel([0.103760, -1.359383, -2.588005, -0.765001, 1.570796, 1.674557],accel_mss,speed_ms,0,blend_radius_m)
    movel([0.103212, -1.359383, -2.588005, -0.765001, 1.570796, 1.674008],accel_mss,speed_ms,0,blend_radius_m)
    movel([0.102701, -1.359360, -2.588021, -0.765008, 1.570796, 1.673497],accel_mss,speed_ms,0,blend_radius_m)
    movel([0.102202, -1.359311, -2.588053, -0.765024, 1.570796, 1.672999],accel_mss,speed_ms,0,blend_radius_m)
    movel([0.101717, -1.359238, -2.588103, -0.765048, 1.570796, 1.672513],accel_mss,speed_ms,0,blend_radius_m)
    movel([0.101237, -1.359139, -2.588170, -0.765080, 1.570796, 1.672033],accel_mss,speed_ms,0,blend_radius_m)
    movel([0.100728, -1.359004, -2.588261, -0.765124, 1.570796, 1.671524],accel_mss,speed_ms,0,blend_radius_m)
    movel([0.100237, -1.358842, -2.588370, -0.765177, 1.570796, 1.671034],accel_mss,speed_ms,0,blend_radius_m)
    movel([0.099800, -1.358662, -2.588492, -0.765236, 1.570796, 1.670597],accel_mss,speed_ms,0,blend_radius_m)
    movel([0.099384, -1.358457, -2.588630, -0.765302, 1.570796, 1.670180],accel_mss,speed_ms,0,blend_radius_m)
    movel([0.099020, -1.358238, -2.588777, -0.765374, 1.570796, 1.669817],accel_mss,speed_ms,0,blend_radius_m)
    movel([0.098775, -1.358054, -2.588901, -0.765434, 1.570796, 1.669571],accel_mss,speed_ms,0,blend_radius_m)
    movel([0.098545, -1.357821, -2.589058, -0.765510, 1.570796, 1.669341],accel_mss,speed_ms,0,blend_radius_m)
    movel([0.098351, -1.357559, -2.589234, -0.765596, 1.570796, 1.669147],accel_mss,speed_ms,0,blend_radius_m)
    movel([0.098188, -1.357254, -2.589439, -0.765696, 1.570796, 1.668985],accel_mss,speed_ms,0,blend_radius_m)
    movel([0.098074, -1.356919, -2.589664, -0.765806, 1.570796, 1.668871],accel_mss,speed_ms,0,blend_radius_m)
    movel([0.098004, -1.356545, -2.589916, -0.765929, 1.570796, 1.668801],accel_mss,speed_ms,0,blend_radius_m)
    movel([0.097972, -1.356122, -2.590199, -0.766068, 1.570796, 1.668769],accel_mss,speed_ms,0,blend_radius_m)
    movel([0.097987, -1.355660, -2.590509, -0.766220, 1.570796, 1.668783],accel_mss,speed_ms,0,blend_radius_m)
    movel([0.098044, -1.355224, -2.590801, -0.766364, 1.570796, 1.668840],accel_mss,speed_ms,0,blend_radius_m)
    movel([0.098105, -1.354951, -2.590983, -0.766454, 1.570796, 1.668901],accel_mss,speed_ms,0,blend_radius_m)
    movel([0.098181, -1.354677, -2.591167, -0.766545, 1.570796, 1.668977],accel_mss,speed_ms,0,blend_radius_m)
    movel([0.098380, -1.354333, -2.591397, -0.766659, 1.570796, 1.669176],accel_mss,speed_ms,0,blend_radius_m)
    movel([0.098617, -1.354134, -2.591529, -0.766725, 1.570796, 1.669414],accel_mss,speed_ms,0,blend_radius_m)
    movel([0.098975, -1.353977, -2.591635, -0.766778, 1.570796, 1.669772],accel_mss,speed_ms,0,blend_radius_m)
    movel([0.099661, -1.353818, -2.591740, -0.766830, 1.570796, 1.670458],accel_mss,speed_ms,0,blend_radius_m)
    movel([0.102034, -1.353283, -2.592097, -0.767009, 1.570796, 1.672831],accel_mss,speed_ms,0,blend_radius_m)
    movel([0.104178, -1.352833, -2.592397, -0.767159, 1.570796, 1.674974],accel_mss,speed_ms,0,blend_radius_m)
    movel([0.113737, -1.350972, -2.593634, -0.767783, 1.570796, 1.684533],accel_mss,speed_ms,0,blend_radius_m)
    movel([0.113991, -1.350939, -2.593656, -0.767794, 1.570796, 1.684787],accel_mss,speed_ms,0,blend_radius_m)
    movel([0.113996, -1.351165, -2.593506, -0.767718, 1.570796, 1.684793],accel_mss,speed_ms,0,blend_radius_m)
    movel([0.113949, -1.352021, -2.592937, -0.767431, 1.570796, 1.684746],accel_mss,speed_ms,0,blend_radius_m)
    movel([0.113889, -1.352751, -2.592452, -0.767186, 1.570796, 1.684685],accel_mss,speed_ms,0,blend_radius_m)
    movel([0.113767, -1.353803, -2.591750, -0.766836, 1.570796, 1.684563],accel_mss,speed_ms,0,blend_radius_m)
    movel([0.113343, -1.357076, -2.589559, -0.765754, 1.570796, 1.684139],accel_mss,speed_ms,0,blend_radius_m)
    movel([0.111877, -1.357671, -2.589159, -0.765559, 1.570796, 1.682674],accel_mss,speed_ms,0,blend_radius_m)
    movel([0.111877, -1.324726, -2.573231, -0.814432, 1.570796, 1.682674],accel_mss,speed_ms,0,blend_radius_m)
    speed_ms = 1.000
    movel([0.102234, -1.319651, -2.576467, -0.816271, 1.570796, 1.673031],accel_mss,speed_ms,0,blend_radius_m)
    speed_ms = 0.008
    movel([0.102234, -1.346471, -2.589611, -0.776307, 1.570796, 1.673031],accel_mss,speed_ms,0,blend_radius_m)
    speed_ms = 0.003
    movel([0.102234, -1.349860, -2.591177, -0.771352, 1.570796, 1.673031],accel_mss,speed_ms,0,blend_radius_m)
    speed_ms = 0.008
    movel([0.100887, -1.350126, -2.591000, -0.771262, 1.570796, 1.671683],accel_mss,speed_ms,0,blend_radius_m)
    movel([0.099931, -1.350301, -2.590884, -0.771204, 1.570796, 1.670727],accel_mss,speed_ms,0,blend_radius_m)
    movel([0.098694, -1.350505, -2.590749, -0.771135, 1.570796, 1.669490],accel_mss,speed_ms,0,blend_radius_m)
    movel([0.100451, -1.349975, -2.591101, -0.771313, 1.570796, 1.671248],accel_mss,speed_ms,0,blend_radius_m)
    movel([0.101949, -1.349648, -2.591317, -0.771424, 1.570796, 1.672745],accel_mss,speed_ms,0,blend_radius_m)
    movel([0.103346, -1.349363, -2.591506, -0.771520, 1.570796, 1.674143],accel_mss,speed_ms,0,blend_radius_m)
    movel([0.104580, -1.349132, -2.591659, -0.771598, 1.570796, 1.675376],accel_mss,speed_ms,0,blend_radius_m)
    movel([0.106093, -1.348887, -2.591821, -0.771681, 1.570796, 1.676890],accel_mss,speed_ms,0,blend_radius_m)
    movel([0.105807, -1.349060, -2.591707, -0.771622, 1.570796, 1.676604],accel_mss,speed_ms,0,blend_radius_m)
    movel([0.104077, -1.349467, -2.591437, -0.771485, 1.570796, 1.674873],accel_mss,speed_ms,0,blend_radius_m)
    movel([0.102234, -1.349860, -2.591177, -0.771352, 1.570796, 1.673031],accel_mss,speed_ms,0,blend_radius_m)
    movel([0.102234, -1.352710, -2.592479, -0.767200, 1.570796, 1.673031],accel_mss,speed_ms,0,blend_radius_m)
    movel([0.100887, -1.352976, -2.592302, -0.767111, 1.570796, 1.671683],accel_mss,speed_ms,0,blend_radius_m)
    movel([0.099931, -1.353150, -2.592186, -0.767053, 1.570796, 1.670727],accel_mss,speed_ms,0,blend_radius_m)
    movel([0.098694, -1.353354, -2.592050, -0.766985, 1.570796, 1.669490],accel_mss,speed_ms,0,blend_radius_m)
    movel([0.100451, -1.352825, -2.592402, -0.767162, 1.570796, 1.671248],accel_mss,speed_ms,0,blend_radius_m)
    movel([0.101949, -1.352499, -2.592619, -0.767271, 1.570796, 1.672745],accel_mss,speed_ms,0,blend_radius_m)
    movel([0.103346, -1.352215, -2.592808, -0.767366, 1.570796, 1.674143],accel_mss,speed_ms,0,blend_radius_m)
    movel([0.104580, -1.351984, -2.592962, -0.767443, 1.570796, 1.675376],accel_mss,speed_ms,0,blend_radius_m)
    movel([0.106093, -1.351739, -2.593125, -0.767525, 1.570796, 1.676890],accel_mss,speed_ms,0,blend_radius_m)
    movel([0.105807, -1.351912, -2.593010, -0.767467, 1.570796, 1.676604],accel_mss,speed_ms,0,blend_radius_m)
    movel([0.104077, -1.352318, -2.592740, -0.767331, 1.570796, 1.674873],accel_mss,speed_ms,0,blend_radius_m)
    movel([0.102234, -1.352710, -2.592479, -0.767200, 1.570796, 1.673031],accel_mss,speed_ms,0,blend_radius_m)
    movel([0.102234, -1.319651, -2.576467, -0.816271, 1.570796, 1.673031],accel_mss,speed_ms,0,blend_radius_m)
    speed_ms = 1.000
    movel([0.134423, -1.321411, -2.575349, -0.815630, 1.570796, 1.705220],accel_mss,speed_ms,0,blend_radius_m)
    speed_ms = 0.008
    movel([0.134423, -1.348200, -2.588469, -0.775720, 1.570796, 1.705220],accel_mss,speed_ms,0,blend_radius_m)
    speed_ms = 0.003
    movel([0.134423, -1.351584, -2.590032, -0.770773, 1.570796, 1.705220],accel_mss,speed_ms,0,blend_radius_m)
    speed_ms = 0.008
    movel([0.134066, -1.351657, -2.589983, -0.770749, 1.570796, 1.704862],accel_mss,speed_ms,0,blend_radius_m)
    movel([0.135260, -1.351288, -2.590229, -0.770872, 1.570796, 1.706056],accel_mss,speed_ms,0,blend_radius_m)
    movel([0.138862, -1.350333, -2.590863, -0.771193, 1.570796, 1.709658],accel_mss,speed_ms,0,blend_radius_m)
    movel([0.142211, -1.349467, -2.591437, -0.771485, 1.570796, 1.713007],accel_mss,speed_ms,0,blend_radius_m)
    movel([0.143351, -1.349189, -2.591621, -0.771579, 1.570796, 1.714147],accel_mss,speed_ms,0,blend_radius_m)
    movel([0.142807, -1.349385, -2.591492, -0.771512, 1.570796, 1.713604],accel_mss,speed_ms,0,blend_radius_m)
    movel([0.140107, -1.350118, -2.591006, -0.771265, 1.570796, 1.710903],accel_mss,speed_ms,0,blend_radius_m)
    movel([0.136916, -1.350954, -2.590451, -0.770984, 1.570796, 1.707712],accel_mss,speed_ms,0,blend_radius_m)
    movel([0.134423, -1.351584, -2.590032, -0.770773, 1.570796, 1.705220],accel_mss,speed_ms,0,blend_radius_m)
    movel([0.134423, -1.354431, -2.591331, -0.766627, 1.570796, 1.705220],accel_mss,speed_ms,0,blend_radius_m)
    movel([0.134066, -1.354503, -2.591283, -0.766603, 1.570796, 1.704862],accel_mss,speed_ms,0,blend_radius_m)
    movel([0.135260, -1.354136, -2.591528, -0.766725, 1.570796, 1.706056],accel_mss,speed_ms,0,blend_radius_m)
    movel([0.138862, -1.353183, -2.592164, -0.767042, 1.570796, 1.709658],accel_mss,speed_ms,0,blend_radius_m)
    movel([0.142211, -1.352318, -2.592740, -0.767331, 1.570796, 1.713007],accel_mss,speed_ms,0,blend_radius_m)
    movel([0.143351, -1.352041, -2.592924, -0.767424, 1.570796, 1.714147],accel_mss,speed_ms,0,blend_radius_m)
    movel([0.142807, -1.352236, -2.592794, -0.767358, 1.570796, 1.713604],accel_mss,speed_ms,0,blend_radius_m)
    movel([0.140107, -1.352968, -2.592307, -0.767114, 1.570796, 1.710903],accel_mss,speed_ms,0,blend_radius_m)
    movel([0.136916, -1.353802, -2.591751, -0.766836, 1.570796, 1.707712],accel_mss,speed_ms,0,blend_radius_m)
    movel([0.134423, -1.354431, -2.591331, -0.766627, 1.570796, 1.705220],accel_mss,speed_ms,0,blend_radius_m)
    movel([0.134423, -1.321411, -2.575349, -0.815630, 1.570796, 1.705220],accel_mss,speed_ms,0,blend_radius_m)
    speed_ms = 1.000
    movel([0.138790, -1.318689, -2.577077, -0.816624, 1.570796, 1.709586],accel_mss,speed_ms,0,blend_radius_m)
    speed_ms = 0.008
    movel([0.138790, -1.345526, -2.590234, -0.776629, 1.570796, 1.709586],accel_mss,speed_ms,0,blend_radius_m)
    speed_ms = 0.003
    movel([0.138790, -1.348917, -2.591801, -0.771671, 1.570796, 1.709586],accel_mss,speed_ms,0,blend_radius_m)
    speed_ms = 0.008
    movel([0.134894, -1.349926, -2.591133, -0.771330, 1.570796, 1.705691],accel_mss,speed_ms,0,blend_radius_m)
    movel([0.132467, -1.350520, -2.590739, -0.771130, 1.570796, 1.703263],accel_mss,speed_ms,0,blend_radius_m)
    movel([0.130576, -1.350959, -2.590447, -0.770983, 1.570796, 1.701372],accel_mss,speed_ms,0,blend_radius_m)
    movel([0.130565, -1.350730, -2.590600, -0.771060, 1.570796, 1.701362],accel_mss,speed_ms,0,blend_radius_m)
    movel([0.132729, -1.350062, -2.591043, -0.771284, 1.570796, 1.703525],accel_mss,speed_ms,0,blend_radius_m)
    movel([0.135050, -1.349395, -2.591485, -0.771509, 1.570796, 1.705846],accel_mss,speed_ms,0,blend_radius_m)
    movel([0.138877, -1.348366, -2.592165, -0.771857, 1.570796, 1.709673],accel_mss,speed_ms,0,blend_radius_m)
    movel([0.142697, -1.347385, -2.592814, -0.772191, 1.570796, 1.713494],accel_mss,speed_ms,0,blend_radius_m)
    movel([0.145007, -1.346834, -2.593176, -0.772378, 1.570796, 1.715803],accel_mss,speed_ms,0,blend_radius_m)
    movel([0.147100, -1.346370, -2.593482, -0.772537, 1.570796, 1.717896],accel_mss,speed_ms,0,blend_radius_m)
    movel([0.147160, -1.346560, -2.593357, -0.772472, 1.570796, 1.717956],accel_mss,speed_ms,0,blend_radius_m)
    movel([0.145142, -1.347190, -2.592942, -0.772257, 1.570796, 1.715938],accel_mss,speed_ms,0,blend_radius_m)
    movel([0.142692, -1.347878, -2.592488, -0.772023, 1.570796, 1.713488],accel_mss,speed_ms,0,blend_radius_m)
    movel([0.138790, -1.348917, -2.591801, -0.771671, 1.570796, 1.709586],accel_mss,speed_ms,0,blend_radius_m)
    movel([0.138790, -1.351770, -2.593104, -0.767515, 1.570796, 1.709586],accel_mss,speed_ms,0,blend_radius_m)
    movel([0.134894, -1.352777, -2.592435, -0.767178, 1.570796, 1.705691],accel_mss,speed_ms,0,blend_radius_m)
    movel([0.132467, -1.353369, -2.592040, -0.766980, 1.570796, 1.703263],accel_mss,speed_ms,0,blend_radius_m)
    movel([0.130576, -1.353807, -2.591748, -0.766834, 1.570796, 1.701372],accel_mss,speed_ms,0,blend_radius_m)
    movel([0.130565, -1.353578, -2.591900, -0.766910, 1.570796, 1.701362],accel_mss,speed_ms,0,blend_radius_m)
    movel([0.132729, -1.352912, -2.592344, -0.767132, 1.570796, 1.703525],accel_mss,speed_ms,0,blend_radius_m)
    movel([0.135050, -1.352247, -2.592787, -0.767355, 1.570796, 1.705846],accel_mss,speed_ms,0,blend_radius_m)
    movel([0.138877, -1.351220, -2.593469, -0.767699, 1.570796, 1.709673],accel_mss,speed_ms,0,blend_radius_m)
    movel([0.142697, -1.350241, -2.594119, -0.768030, 1.570796, 1.713494],accel_mss,speed_ms,0,blend_radius_m)
    movel([0.145007, -1.349691, -2.594482, -0.768215, 1.570796, 1.715803],accel_mss,speed_ms,0,blend_radius_m)
    movel([0.147100, -1.349228, -2.594789, -0.768372, 1.570796, 1.717896],accel_mss,speed_ms,0,blend_radius_m)
    movel([0.147160, -1.349418, -2.594663, -0.768308, 1.570796, 1.717956],accel_mss,speed_ms,0,blend_radius_m)
    movel([0.145142, -1.350047, -2.594247, -0.768095, 1.570796, 1.715938],accel_mss,speed_ms,0,blend_radius_m)
    movel([0.142692, -1.350733, -2.593793, -0.767864, 1.570796, 1.713488],accel_mss,speed_ms,0,blend_radius_m)
    movel([0.138790, -1.351770, -2.593104, -0.767515, 1.570796, 1.709586],accel_mss,speed_ms,0,blend_radius_m)
    movel([0.138790, -1.318689, -2.577077, -0.816624, 1.570796, 1.709586],accel_mss,speed_ms,0,blend_radius_m)
    speed_ms = 1.000
    movel([0.139206, -1.316958, -2.578170, -0.817261, 1.570796, 1.710002],accel_mss,speed_ms,0,blend_radius_m)
    speed_ms = 0.008
    movel([0.139206, -1.343827, -2.591350, -0.777212, 1.570796, 1.710002],accel_mss,speed_ms,0,blend_radius_m)
    speed_ms = 0.003
    movel([0.139206, -1.347222, -2.592921, -0.772246, 1.570796, 1.710002],accel_mss,speed_ms,0,blend_radius_m)
    speed_ms = 0.008
    movel([0.114266, -1.354008, -2.588415, -0.769966, 1.570796, 1.685062],accel_mss,speed_ms,0,blend_radius_m)
    movel([0.121316, -1.301208, -2.621827, -0.789355, 1.570796, 1.692112],accel_mss,speed_ms,0,blend_radius_m)
    movel([0.174540, -1.286058, -2.630734, -0.795597, 1.570796, 1.745336],accel_mss,speed_ms,0,blend_radius_m)
    movel([0.164255, -1.340855, -2.597091, -0.774443, 1.570796, 1.735051],accel_mss,speed_ms,0,blend_radius_m)
    movel([0.139206, -1.347222, -2.592921, -0.772246, 1.570796, 1.710002],accel_mss,speed_ms,0,blend_radius_m)
    movel([0.139206, -1.350078, -2.594226, -0.768084, 1.570796, 1.710002],accel_mss,speed_ms,0,blend_radius_m)
    movel([0.114266, -1.356850, -2.589711, -0.765828, 1.570796, 1.685062],accel_mss,speed_ms,0,blend_radius_m)
    movel([0.121316, -1.304157, -2.623198, -0.785034, 1.570796, 1.692112],accel_mss,speed_ms,0,blend_radius_m)
    movel([0.174540, -1.289036, -2.632127, -0.791226, 1.570796, 1.745336],accel_mss,speed_ms,0,blend_radius_m)
    movel([0.164255, -1.343725, -2.598405, -0.770259, 1.570796, 1.735051],accel_mss,speed_ms,0,blend_radius_m)
    movel([0.139206, -1.350078, -2.594226, -0.768084, 1.570796, 1.710002],accel_mss,speed_ms,0,blend_radius_m)
    movel([0.139206, -1.316958, -2.578170, -0.817261, 1.570796, 1.710002],accel_mss,speed_ms,0,blend_radius_m)
    speed_ms = 1.000
    movel([0.146479, -1.328997, -2.570482, -0.812910, 1.570796, 1.717275],accel_mss,speed_ms,0,blend_radius_m)
    speed_ms = 0.008
    movel([0.146479, -1.355648, -2.583500, -0.773241, 1.570796, 1.717275],accel_mss,speed_ms,0,blend_radius_m)
    speed_ms = 0.003
    movel([0.146479, -1.359013, -2.585051, -0.768325, 1.570796, 1.717275],accel_mss,speed_ms,0,blend_radius_m)
    speed_ms = 0.008
    movel([0.145933, -1.358974, -2.585077, -0.768338, 1.570796, 1.716730],accel_mss,speed_ms,0,blend_radius_m)
    movel([0.145377, -1.358954, -2.585091, -0.768344, 1.570796, 1.716173],accel_mss,speed_ms,0,blend_radius_m)
    movel([0.144812, -1.358955, -2.585090, -0.768344, 1.570796, 1.715609],accel_mss,speed_ms,0,blend_radius_m)
    movel([0.144237, -1.358977, -2.585075, -0.768337, 1.570796, 1.715033],accel_mss,speed_ms,0,blend_radius_m)
    movel([0.143671, -1.359016, -2.585049, -0.768324, 1.570796, 1.714467],accel_mss,speed_ms,0,blend_radius_m)
    movel([0.143096, -1.359075, -2.585009, -0.768305, 1.570796, 1.713893],accel_mss,speed_ms,0,blend_radius_m)
    movel([0.142574, -1.359145, -2.584962, -0.768282, 1.570796, 1.713370],accel_mss,speed_ms,0,blend_radius_m)
    movel([0.141799, -1.359266, -2.584880, -0.768243, 1.570796, 1.712595],accel_mss,speed_ms,0,blend_radius_m)
    movel([0.140898, -1.359422, -2.584774, -0.768193, 1.570796, 1.711695],accel_mss,speed_ms,0,blend_radius_m)
    movel([0.140000, -1.359596, -2.584657, -0.768136, 1.570796, 1.710796],accel_mss,speed_ms,0,blend_radius_m)
    movel([0.139097, -1.359786, -2.584528, -0.768075, 1.570796, 1.709893],accel_mss,speed_ms,0,blend_radius_m)
    movel([0.138186, -1.359992, -2.584388, -0.768008, 1.570796, 1.708983],accel_mss,speed_ms,0,blend_radius_m)
    movel([0.137270, -1.360220, -2.584234, -0.767935, 1.570796, 1.708066],accel_mss,speed_ms,0,blend_radius_m)
    movel([0.136360, -1.360460, -2.584072, -0.767857, 1.570796, 1.707156],accel_mss,speed_ms,0,blend_radius_m)
    movel([0.135446, -1.360718, -2.583897, -0.767774, 1.570796, 1.706243],accel_mss,speed_ms,0,blend_radius_m)
    movel([0.134526, -1.360992, -2.583711, -0.767686, 1.570796, 1.705323],accel_mss,speed_ms,0,blend_radius_m)
    movel([0.133629, -1.361277, -2.583517, -0.767594, 1.570796, 1.704426],accel_mss,speed_ms,0,blend_radius_m)
    movel([0.132730, -1.361577, -2.583314, -0.767498, 1.570796, 1.703527],accel_mss,speed_ms,0,blend_radius_m)
    movel([0.131749, -1.361922, -2.583079, -0.767388, 1.570796, 1.702545],accel_mss,speed_ms,0,blend_radius_m)
    movel([0.131133, -1.362153, -2.582923, -0.767314, 1.570796, 1.701929],accel_mss,speed_ms,0,blend_radius_m)
    movel([0.130482, -1.362419, -2.582742, -0.767229, 1.570796, 1.701278],accel_mss,speed_ms,0,blend_radius_m)
    movel([0.129833, -1.362703, -2.582548, -0.767138, 1.570796, 1.700630],accel_mss,speed_ms,0,blend_radius_m)
    movel([0.129187, -1.363009, -2.582339, -0.767040, 1.570796, 1.699983],accel_mss,speed_ms,0,blend_radius_m)
    movel([0.128546, -1.363331, -2.582120, -0.766938, 1.570796, 1.699342],accel_mss,speed_ms,0,blend_radius_m)
    movel([0.128002, -1.363621, -2.581922, -0.766845, 1.570796, 1.698799],accel_mss,speed_ms,0,blend_radius_m)
    movel([0.127491, -1.363909, -2.581726, -0.766754, 1.570796, 1.698288],accel_mss,speed_ms,0,blend_radius_m)
    movel([0.127184, -1.364107, -2.581591, -0.766691, 1.570796, 1.697980],accel_mss,speed_ms,0,blend_radius_m)
    movel([0.126843, -1.364420, -2.581377, -0.766592, 1.570796, 1.697639],accel_mss,speed_ms,0,blend_radius_m)
    movel([0.126700, -1.364750, -2.581151, -0.766487, 1.570796, 1.697496],accel_mss,speed_ms,0,blend_radius_m)
    movel([0.126658, -1.365077, -2.580928, -0.766384, 1.570796, 1.697454],accel_mss,speed_ms,0,blend_radius_m)
    movel([0.126664, -1.365455, -2.580669, -0.766265, 1.570796, 1.697460],accel_mss,speed_ms,0,blend_radius_m)
    movel([0.126770, -1.365766, -2.580456, -0.766167, 1.570796, 1.697566],accel_mss,speed_ms,0,blend_radius_m)
    movel([0.126938, -1.365865, -2.580388, -0.766136, 1.570796, 1.697735],accel_mss,speed_ms,0,blend_radius_m)
    movel([0.127195, -1.365842, -2.580404, -0.766143, 1.570796, 1.697992],accel_mss,speed_ms,0,blend_radius_m)
    movel([0.127527, -1.365759, -2.580461, -0.766169, 1.570796, 1.698323],accel_mss,speed_ms,0,blend_radius_m)
    movel([0.127863, -1.365645, -2.580539, -0.766205, 1.570796, 1.698659],accel_mss,speed_ms,0,blend_radius_m)
    movel([0.131526, -1.364207, -2.581522, -0.766659, 1.570796, 1.702322],accel_mss,speed_ms,0,blend_radius_m)
    movel([0.132241, -1.363941, -2.581704, -0.766744, 1.570796, 1.703038],accel_mss,speed_ms,0,blend_radius_m)
    movel([0.132957, -1.363690, -2.581875, -0.766824, 1.570796, 1.703754],accel_mss,speed_ms,0,blend_radius_m)
    movel([0.133827, -1.363410, -2.582066, -0.766912, 1.570796, 1.704623],accel_mss,speed_ms,0,blend_radius_m)
    movel([0.134786, -1.363123, -2.582262, -0.767004, 1.570796, 1.705582],accel_mss,speed_ms,0,blend_radius_m)
    movel([0.135920, -1.362806, -2.582478, -0.767105, 1.570796, 1.706717],accel_mss,speed_ms,0,blend_radius_m)
    movel([0.137052, -1.362508, -2.582681, -0.767200, 1.570796, 1.707849],accel_mss,speed_ms,0,blend_radius_m)
    movel([0.138308, -1.362203, -2.582888, -0.767298, 1.570796, 1.709104],accel_mss,speed_ms,0,blend_radius_m)
    movel([0.139555, -1.361923, -2.583079, -0.767387, 1.570796, 1.710351],accel_mss,speed_ms,0,blend_radius_m)
    movel([0.140813, -1.361667, -2.583253, -0.767469, 1.570796, 1.711609],accel_mss,speed_ms,0,blend_radius_m)
    movel([0.141996, -1.361450, -2.583400, -0.767539, 1.570796, 1.712793],accel_mss,speed_ms,0,blend_radius_m)
    movel([0.142726, -1.361341, -2.583474, -0.767574, 1.570796, 1.713523],accel_mss,speed_ms,0,blend_radius_m)
    movel([0.143450, -1.361255, -2.583532, -0.767601, 1.570796, 1.714246],accel_mss,speed_ms,0,blend_radius_m)
    movel([0.144051, -1.361201, -2.583569, -0.767619, 1.570796, 1.714848],accel_mss,speed_ms,0,blend_radius_m)
    movel([0.145020, -1.361135, -2.583614, -0.767640, 1.570796, 1.715817],accel_mss,speed_ms,0,blend_radius_m)
    movel([0.145558, -1.361084, -2.583648, -0.767656, 1.570796, 1.716354],accel_mss,speed_ms,0,blend_radius_m)
    movel([0.146191, -1.361001, -2.583705, -0.767683, 1.570796, 1.716987],accel_mss,speed_ms,0,blend_radius_m)
    movel([0.146473, -1.360957, -2.583735, -0.767697, 1.570796, 1.717270],accel_mss,speed_ms,0,blend_radius_m)
    movel([0.146735, -1.360790, -2.583848, -0.767751, 1.570796, 1.717531],accel_mss,speed_ms,0,blend_radius_m)
    movel([0.146899, -1.360434, -2.584089, -0.767866, 1.570796, 1.717695],accel_mss,speed_ms,0,blend_radius_m)
    movel([0.146972, -1.360199, -2.584248, -0.767941, 1.570796, 1.717769],accel_mss,speed_ms,0,blend_radius_m)
    movel([0.147032, -1.359929, -2.584431, -0.768029, 1.570796, 1.717828],accel_mss,speed_ms,0,blend_radius_m)
    movel([0.147067, -1.359499, -2.584722, -0.768168, 1.570796, 1.717863],accel_mss,speed_ms,0,blend_radius_m)
    movel([0.147027, -1.359301, -2.584856, -0.768232, 1.570796, 1.717823],accel_mss,speed_ms,0,blend_radius_m)
    movel([0.146840, -1.359105, -2.584989, -0.768295, 1.570796, 1.717636],accel_mss,speed_ms,0,blend_radius_m)
    movel([0.146479, -1.359013, -2.585051, -0.768325, 1.570796, 1.717275],accel_mss,speed_ms,0,blend_radius_m)
    movel([0.146479, -1.361844, -2.586340, -0.764206, 1.570796, 1.717275],accel_mss,speed_ms,0,blend_radius_m)
    movel([0.145933, -1.361805, -2.586366, -0.764218, 1.570796, 1.716730],accel_mss,speed_ms,0,blend_radius_m)
    movel([0.145377, -1.361784, -2.586380, -0.764225, 1.570796, 1.716173],accel_mss,speed_ms,0,blend_radius_m)
    movel([0.144812, -1.361786, -2.586379, -0.764224, 1.570796, 1.715609],accel_mss,speed_ms,0,blend_radius_m)
    movel([0.144237, -1.361807, -2.586364, -0.764217, 1.570796, 1.715033],accel_mss,speed_ms,0,blend_radius_m)
    movel([0.143671, -1.361847, -2.586338, -0.764205, 1.570796, 1.714467],accel_mss,speed_ms,0,blend_radius_m)
    movel([0.143096, -1.361905, -2.586298, -0.764186, 1.570796, 1.713893],accel_mss,speed_ms,0,blend_radius_m)
    movel([0.142574, -1.361975, -2.586251, -0.764163, 1.570796, 1.713370],accel_mss,speed_ms,0,blend_radius_m)
    movel([0.141799, -1.362096, -2.586168, -0.764125, 1.570796, 1.712595],accel_mss,speed_ms,0,blend_radius_m)
    movel([0.140898, -1.362252, -2.586063, -0.764075, 1.570796, 1.711695],accel_mss,speed_ms,0,blend_radius_m)
    movel([0.140000, -1.362425, -2.585945, -0.764019, 1.570796, 1.710796],accel_mss,speed_ms,0,blend_radius_m)
    movel([0.139097, -1.362615, -2.585816, -0.763958, 1.570796, 1.709893],accel_mss,speed_ms,0,blend_radius_m)
    movel([0.138186, -1.362821, -2.585676, -0.763892, 1.570796, 1.708983],accel_mss,speed_ms,0,blend_radius_m)
    movel([0.137270, -1.363048, -2.585521, -0.763820, 1.570796, 1.708066],accel_mss,speed_ms,0,blend_radius_m)
    movel([0.136360, -1.363287, -2.585359, -0.763743, 1.570796, 1.707156],accel_mss,speed_ms,0,blend_radius_m)
    movel([0.135446, -1.363545, -2.585183, -0.763661, 1.570796, 1.706243],accel_mss,speed_ms,0,blend_radius_m)
    movel([0.134526, -1.363818, -2.584997, -0.763574, 1.570796, 1.705323],accel_mss,speed_ms,0,blend_radius_m)
    movel([0.133629, -1.364103, -2.584803, -0.763483, 1.570796, 1.704426],accel_mss,speed_ms,0,blend_radius_m)
    movel([0.132730, -1.364402, -2.584599, -0.763388, 1.570796, 1.703527],accel_mss,speed_ms,0,blend_radius_m)
    movel([0.131749, -1.364746, -2.584364, -0.763279, 1.570796, 1.702545],accel_mss,speed_ms,0,blend_radius_m)
    movel([0.131133, -1.364976, -2.584207, -0.763206, 1.570796, 1.701929],accel_mss,speed_ms,0,blend_radius_m)
    movel([0.130482, -1.365242, -2.584026, -0.763122, 1.570796, 1.701278],accel_mss,speed_ms,0,blend_radius_m)
    movel([0.129833, -1.365526, -2.583832, -0.763032, 1.570796, 1.700630],accel_mss,speed_ms,0,blend_radius_m)
    movel([0.129187, -1.365831, -2.583623, -0.762935, 1.570796, 1.699983],accel_mss,speed_ms,0,blend_radius_m)
    movel([0.128546, -1.366152, -2.583403, -0.762834, 1.570796, 1.699342],accel_mss,speed_ms,0,blend_radius_m)
    movel([0.128002, -1.366442, -2.583205, -0.762743, 1.570796, 1.698799],accel_mss,speed_ms,0,blend_radius_m)
    movel([0.127491, -1.366729, -2.583008, -0.762652, 1.570796, 1.698288],accel_mss,speed_ms,0,blend_radius_m)
    movel([0.127184, -1.366926, -2.582873, -0.762590, 1.570796, 1.697980],accel_mss,speed_ms,0,blend_radius_m)
    movel([0.126843, -1.367239, -2.582658, -0.762492, 1.570796, 1.697639],accel_mss,speed_ms,0,blend_radius_m)
    movel([0.126700, -1.367568, -2.582432, -0.762389, 1.570796, 1.697496],accel_mss,speed_ms,0,blend_radius_m)
    movel([0.126658, -1.367894, -2.582208, -0.762287, 1.570796, 1.697454],accel_mss,speed_ms,0,blend_radius_m)
    movel([0.126664, -1.368272, -2.581949, -0.762169, 1.570796, 1.697460],accel_mss,speed_ms,0,blend_radius_m)
    movel([0.126770, -1.368582, -2.581735, -0.762072, 1.570796, 1.697566],accel_mss,speed_ms,0,blend_radius_m)
    movel([0.126938, -1.368681, -2.581667, -0.762041, 1.570796, 1.697735],accel_mss,speed_ms,0,blend_radius_m)
    movel([0.127195, -1.368658, -2.581683, -0.762048, 1.570796, 1.697992],accel_mss,speed_ms,0,blend_radius_m)
    movel([0.127527, -1.368575, -2.581740, -0.762074, 1.570796, 1.698323],accel_mss,speed_ms,0,blend_radius_m)
    movel([0.127863, -1.368461, -2.581819, -0.762110, 1.570796, 1.698659],accel_mss,speed_ms,0,blend_radius_m)
    movel([0.131526, -1.367027, -2.582804, -0.762559, 1.570796, 1.702322],accel_mss,speed_ms,0,blend_radius_m)
    movel([0.132241, -1.366761, -2.582986, -0.762642, 1.570796, 1.703038],accel_mss,speed_ms,0,blend_radius_m)
    movel([0.132957, -1.366510, -2.583158, -0.762721, 1.570796, 1.703754],accel_mss,speed_ms,0,blend_radius_m)
    movel([0.133827, -1.366231, -2.583349, -0.762809, 1.570796, 1.704623],accel_mss,speed_ms,0,blend_radius_m)
    movel([0.134786, -1.365945, -2.583545, -0.762899, 1.570796, 1.705582],accel_mss,speed_ms,0,blend_radius_m)
    movel([0.135920, -1.365628, -2.583761, -0.762999, 1.570796, 1.706717],accel_mss,speed_ms,0,blend_radius_m)
    movel([0.137052, -1.365331, -2.583965, -0.763093, 1.570796, 1.707849],accel_mss,speed_ms,0,blend_radius_m)
    movel([0.138308, -1.365026, -2.584173, -0.763190, 1.570796, 1.709104],accel_mss,speed_ms,0,blend_radius_m)
    movel([0.139555, -1.364747, -2.584364, -0.763278, 1.570796, 1.710351],accel_mss,speed_ms,0,blend_radius_m)
    movel([0.140813, -1.364491, -2.584538, -0.763360, 1.570796, 1.711609],accel_mss,speed_ms,0,blend_radius_m)
    movel([0.141996, -1.364275, -2.584685, -0.763428, 1.570796, 1.712793],accel_mss,speed_ms,0,blend_radius_m)
    movel([0.142726, -1.364166, -2.584760, -0.763463, 1.570796, 1.713523],accel_mss,speed_ms,0,blend_radius_m)
    movel([0.143450, -1.364081, -2.584818, -0.763490, 1.570796, 1.714246],accel_mss,speed_ms,0,blend_radius_m)
    movel([0.144051, -1.364027, -2.584855, -0.763507, 1.570796, 1.714848],accel_mss,speed_ms,0,blend_radius_m)
    movel([0.145020, -1.363961, -2.584900, -0.763528, 1.570796, 1.715817],accel_mss,speed_ms,0,blend_radius_m)
    movel([0.145558, -1.363910, -2.584934, -0.763544, 1.570796, 1.716354],accel_mss,speed_ms,0,blend_radius_m)
    movel([0.146191, -1.363828, -2.584991, -0.763571, 1.570796, 1.716987],accel_mss,speed_ms,0,blend_radius_m)
    movel([0.146473, -1.363783, -2.585021, -0.763585, 1.570796, 1.717270],accel_mss,speed_ms,0,blend_radius_m)
    movel([0.146735, -1.363616, -2.585135, -0.763638, 1.570796, 1.717531],accel_mss,speed_ms,0,blend_radius_m)
    movel([0.146899, -1.363262, -2.585376, -0.763751, 1.570796, 1.717695],accel_mss,speed_ms,0,blend_radius_m)
    movel([0.146972, -1.363027, -2.585535, -0.763826, 1.570796, 1.717769],accel_mss,speed_ms,0,blend_radius_m)
    movel([0.147032, -1.362757, -2.585719, -0.763913, 1.570796, 1.717828],accel_mss,speed_ms,0,blend_radius_m)
    movel([0.147067, -1.362329, -2.586010, -0.764050, 1.570796, 1.717863],accel_mss,speed_ms,0,blend_radius_m)
    movel([0.147027, -1.362131, -2.586145, -0.764113, 1.570796, 1.717823],accel_mss,speed_ms,0,blend_radius_m)
    movel([0.146840, -1.361935, -2.586278, -0.764176, 1.570796, 1.717636],accel_mss,speed_ms,0,blend_radius_m)
    movel([0.146479, -1.361844, -2.586340, -0.764206, 1.570796, 1.717275],accel_mss,speed_ms,0,blend_radius_m)
    movel([0.146479, -1.328997, -2.570482, -0.812910, 1.570796, 1.717275],accel_mss,speed_ms,0,blend_radius_m)
    speed_ms = 1.000
    movel([0.148139, -1.339270, -2.563771, -0.809348, 1.570796, 1.718936],accel_mss,speed_ms,0,blend_radius_m)
    speed_ms = 0.008
    movel([0.148139, -1.365730, -2.576652, -0.770008, 1.570796, 1.718936],accel_mss,speed_ms,0,blend_radius_m)
    speed_ms = 0.003
    movel([0.148139, -1.369069, -2.578185, -0.765135, 1.570796, 1.718936],accel_mss,speed_ms,0,blend_radius_m)
    speed_ms = 0.008
    movel([0.148028, -1.368798, -2.578372, -0.765219, 1.570796, 1.718824],accel_mss,speed_ms,0,blend_radius_m)
    movel([0.147876, -1.368553, -2.578541, -0.765295, 1.570796, 1.718672],accel_mss,speed_ms,0,blend_radius_m)
    movel([0.147690, -1.368335, -2.578691, -0.765363, 1.570796, 1.718487],accel_mss,speed_ms,0,blend_radius_m)
    movel([0.147468, -1.368147, -2.578820, -0.765421, 1.570796, 1.718264],accel_mss,speed_ms,0,blend_radius_m)
    movel([0.147175, -1.367964, -2.578946, -0.765478, 1.570796, 1.717971],accel_mss,speed_ms,0,blend_radius_m)
    movel([0.146851, -1.367817, -2.579048, -0.765524, 1.570796, 1.717647],accel_mss,speed_ms,0,blend_radius_m)
    movel([0.146500, -1.367702, -2.579127, -0.765560, 1.570796, 1.717297],accel_mss,speed_ms,0,blend_radius_m)
    movel([0.146126, -1.367623, -2.579182, -0.765585, 1.570796, 1.716923],accel_mss,speed_ms,0,blend_radius_m)
    movel([0.145734, -1.367582, -2.579209, -0.765597, 1.570796, 1.716530],accel_mss,speed_ms,0,blend_radius_m)
    movel([0.145328, -1.367576, -2.579214, -0.765600, 1.570796, 1.716125],accel_mss,speed_ms,0,blend_radius_m)
    movel([0.144903, -1.367604, -2.579194, -0.765591, 1.570796, 1.715699],accel_mss,speed_ms,0,blend_radius_m)
    movel([0.144479, -1.367664, -2.579153, -0.765572, 1.570796, 1.715275],accel_mss,speed_ms,0,blend_radius_m)
    movel([0.144074, -1.367758, -2.579088, -0.765543, 1.570796, 1.714870],accel_mss,speed_ms,0,blend_radius_m)
    movel([0.143665, -1.367888, -2.578999, -0.765502, 1.570796, 1.714462],accel_mss,speed_ms,0,blend_radius_m)
    movel([0.143256, -1.368050, -2.578888, -0.765452, 1.570796, 1.714053],accel_mss,speed_ms,0,blend_radius_m)
    movel([0.142845, -1.368244, -2.578754, -0.765391, 1.570796, 1.713641],accel_mss,speed_ms,0,blend_radius_m)
    movel([0.142424, -1.368480, -2.578591, -0.765318, 1.570796, 1.713221],accel_mss,speed_ms,0,blend_radius_m)
    movel([0.142012, -1.368741, -2.578411, -0.765236, 1.570796, 1.712808],accel_mss,speed_ms,0,blend_radius_m)
    movel([0.141614, -1.369031, -2.578211, -0.765147, 1.570796, 1.712411],accel_mss,speed_ms,0,blend_radius_m)
    movel([0.141235, -1.369344, -2.577995, -0.765049, 1.570796, 1.712031],accel_mss,speed_ms,0,blend_radius_m)
    movel([0.140877, -1.369677, -2.577765, -0.764946, 1.570796, 1.711673],accel_mss,speed_ms,0,blend_radius_m)
    movel([0.140540, -1.370031, -2.577521, -0.764837, 1.570796, 1.711336],accel_mss,speed_ms,0,blend_radius_m)
    movel([0.140246, -1.370384, -2.577277, -0.764728, 1.570796, 1.711043],accel_mss,speed_ms,0,blend_radius_m)
    movel([0.139986, -1.370746, -2.577026, -0.764617, 1.570796, 1.710782],accel_mss,speed_ms,0,blend_radius_m)
    movel([0.139757, -1.371119, -2.576768, -0.764502, 1.570796, 1.710554],accel_mss,speed_ms,0,blend_radius_m)
    movel([0.139564, -1.371497, -2.576506, -0.764386, 1.570796, 1.710361],accel_mss,speed_ms,0,blend_radius_m)
    movel([0.139410, -1.371875, -2.576244, -0.764270, 1.570796, 1.710206],accel_mss,speed_ms,0,blend_radius_m)
    movel([0.139295, -1.372251, -2.575983, -0.764155, 1.570796, 1.710091],accel_mss,speed_ms,0,blend_radius_m)
    movel([0.139220, -1.372614, -2.575731, -0.764044, 1.570796, 1.710017],accel_mss,speed_ms,0,blend_radius_m)
    movel([0.139188, -1.372969, -2.575484, -0.763936, 1.570796, 1.709984],accel_mss,speed_ms,0,blend_radius_m)
    movel([0.139200, -1.373306, -2.575250, -0.763833, 1.570796, 1.709996],accel_mss,speed_ms,0,blend_radius_m)
    movel([0.139250, -1.373627, -2.575026, -0.763736, 1.570796, 1.710046],accel_mss,speed_ms,0,blend_radius_m)
    movel([0.139348, -1.373936, -2.574811, -0.763642, 1.570796, 1.710144],accel_mss,speed_ms,0,blend_radius_m)
    movel([0.139488, -1.374219, -2.574614, -0.763556, 1.570796, 1.710284],accel_mss,speed_ms,0,blend_radius_m)
    movel([0.139673, -1.374477, -2.574434, -0.763478, 1.570796, 1.710469],accel_mss,speed_ms,0,blend_radius_m)
    movel([0.139898, -1.374707, -2.574274, -0.763409, 1.570796, 1.710695],accel_mss,speed_ms,0,blend_radius_m)
    movel([0.140160, -1.374905, -2.574135, -0.763349, 1.570796, 1.710956],accel_mss,speed_ms,0,blend_radius_m)
    movel([0.140456, -1.375067, -2.574022, -0.763300, 1.570796, 1.711252],accel_mss,speed_ms,0,blend_radius_m)
    movel([0.140782, -1.375194, -2.573934, -0.763262, 1.570796, 1.711578],accel_mss,speed_ms,0,blend_radius_m)
    movel([0.141137, -1.375281, -2.573872, -0.763235, 1.570796, 1.711934],accel_mss,speed_ms,0,blend_radius_m)
    movel([0.141514, -1.375330, -2.573838, -0.763221, 1.570796, 1.712310],accel_mss,speed_ms,0,blend_radius_m)
    movel([0.141920, -1.375342, -2.573830, -0.763217, 1.570796, 1.712716],accel_mss,speed_ms,0,blend_radius_m)
    movel([0.142340, -1.375315, -2.573849, -0.763225, 1.570796, 1.713136],accel_mss,speed_ms,0,blend_radius_m)
    movel([0.142773, -1.375251, -2.573894, -0.763244, 1.570796, 1.713569],accel_mss,speed_ms,0,blend_radius_m)
    movel([0.143214, -1.375149, -2.573965, -0.763275, 1.570796, 1.714011],accel_mss,speed_ms,0,blend_radius_m)
    movel([0.143660, -1.375010, -2.574062, -0.763317, 1.570796, 1.714456],accel_mss,speed_ms,0,blend_radius_m)
    movel([0.144106, -1.374834, -2.574185, -0.763370, 1.570796, 1.714903],accel_mss,speed_ms,0,blend_radius_m)
    movel([0.144549, -1.374626, -2.574330, -0.763433, 1.570796, 1.715345],accel_mss,speed_ms,0,blend_radius_m)
    movel([0.144987, -1.374385, -2.574498, -0.763506, 1.570796, 1.715783],accel_mss,speed_ms,0,blend_radius_m)
    movel([0.145417, -1.374110, -2.574690, -0.763589, 1.570796, 1.716213],accel_mss,speed_ms,0,blend_radius_m)
    movel([0.145830, -1.373810, -2.574899, -0.763680, 1.570796, 1.716626],accel_mss,speed_ms,0,blend_radius_m)
    movel([0.146222, -1.373484, -2.575126, -0.763779, 1.570796, 1.717019],accel_mss,speed_ms,0,blend_radius_m)
    movel([0.146587, -1.373142, -2.575364, -0.763883, 1.570796, 1.717383],accel_mss,speed_ms,0,blend_radius_m)
    movel([0.146918, -1.372787, -2.575611, -0.763991, 1.570796, 1.717715],accel_mss,speed_ms,0,blend_radius_m)
    movel([0.147221, -1.372415, -2.575869, -0.764105, 1.570796, 1.718017],accel_mss,speed_ms,0,blend_radius_m)
    movel([0.147490, -1.372032, -2.576135, -0.764222, 1.570796, 1.718286],accel_mss,speed_ms,0,blend_radius_m)
    movel([0.147725, -1.371633, -2.576412, -0.764344, 1.570796, 1.718521],accel_mss,speed_ms,0,blend_radius_m)
    movel([0.147922, -1.371233, -2.576689, -0.764467, 1.570796, 1.718719],accel_mss,speed_ms,0,blend_radius_m)
    movel([0.148071, -1.370849, -2.576955, -0.764585, 1.570796, 1.718868],accel_mss,speed_ms,0,blend_radius_m)
    movel([0.148177, -1.370467, -2.577220, -0.764703, 1.570796, 1.718973],accel_mss,speed_ms,0,blend_radius_m)
    movel([0.148237, -1.370093, -2.577478, -0.764818, 1.570796, 1.719033],accel_mss,speed_ms,0,blend_radius_m)
    movel([0.148252, -1.369732, -2.577727, -0.764929, 1.570796, 1.719048],accel_mss,speed_ms,0,blend_radius_m)
    movel([0.148218, -1.369390, -2.577964, -0.765035, 1.570796, 1.719014],accel_mss,speed_ms,0,blend_radius_m)
    movel([0.148139, -1.369069, -2.578185, -0.765135, 1.570796, 1.718936],accel_mss,speed_ms,0,blend_radius_m)
    movel([0.148139, -1.371877, -2.579460, -0.761052, 1.570796, 1.718936],accel_mss,speed_ms,0,blend_radius_m)
    movel([0.148028, -1.371607, -2.579647, -0.761135, 1.570796, 1.718824],accel_mss,speed_ms,0,blend_radius_m)
    movel([0.147876, -1.371362, -2.579817, -0.761210, 1.570796, 1.718672],accel_mss,speed_ms,0,blend_radius_m)
    movel([0.147690, -1.371145, -2.579967, -0.761277, 1.570796, 1.718487],accel_mss,speed_ms,0,blend_radius_m)
    movel([0.147468, -1.370958, -2.580096, -0.761335, 1.570796, 1.718264],accel_mss,speed_ms,0,blend_radius_m)
    movel([0.147175, -1.370775, -2.580223, -0.761391, 1.570796, 1.717971],accel_mss,speed_ms,0,blend_radius_m)
    movel([0.146851, -1.370628, -2.580324, -0.761437, 1.570796, 1.717647],accel_mss,speed_ms,0,blend_radius_m)
    movel([0.146500, -1.370513, -2.580404, -0.761472, 1.570796, 1.717297],accel_mss,speed_ms,0,blend_radius_m)
    movel([0.146126, -1.370434, -2.580458, -0.761497, 1.570796, 1.716923],accel_mss,speed_ms,0,blend_radius_m)
    movel([0.145734, -1.370394, -2.580486, -0.761509, 1.570796, 1.716530],accel_mss,speed_ms,0,blend_radius_m)
    movel([0.145328, -1.370387, -2.580491, -0.761511, 1.570796, 1.716125],accel_mss,speed_ms,0,blend_radius_m)
    movel([0.144903, -1.370415, -2.580471, -0.761502, 1.570796, 1.715699],accel_mss,speed_ms,0,blend_radius_m)
    movel([0.144479, -1.370475, -2.580430, -0.761484, 1.570796, 1.715275],accel_mss,speed_ms,0,blend_radius_m)
    movel([0.144074, -1.370569, -2.580365, -0.761455, 1.570796, 1.714870],accel_mss,speed_ms,0,blend_radius_m)
    movel([0.143665, -1.370699, -2.580276, -0.761415, 1.570796, 1.714462],accel_mss,speed_ms,0,blend_radius_m)
    movel([0.143256, -1.370860, -2.580164, -0.761365, 1.570796, 1.714053],accel_mss,speed_ms,0,blend_radius_m)
    movel([0.142845, -1.371054, -2.580030, -0.761305, 1.570796, 1.713641],accel_mss,speed_ms,0,blend_radius_m)
    movel([0.142424, -1.371289, -2.579867, -0.761233, 1.570796, 1.713221],accel_mss,speed_ms,0,blend_radius_m)
    movel([0.142012, -1.371550, -2.579686, -0.761152, 1.570796, 1.712808],accel_mss,speed_ms,0,blend_radius_m)
    movel([0.141614, -1.371839, -2.579486, -0.761063, 1.570796, 1.712411],accel_mss,speed_ms,0,blend_radius_m)
    movel([0.141235, -1.372152, -2.579270, -0.760967, 1.570796, 1.712031],accel_mss,speed_ms,0,blend_radius_m)
    movel([0.140877, -1.372484, -2.579039, -0.760866, 1.570796, 1.711673],accel_mss,speed_ms,0,blend_radius_m)
    movel([0.140540, -1.372837, -2.578795, -0.760758, 1.570796, 1.711336],accel_mss,speed_ms,0,blend_radius_m)
    movel([0.140246, -1.373189, -2.578550, -0.760650, 1.570796, 1.711043],accel_mss,speed_ms,0,blend_radius_m)
    movel([0.139986, -1.373550, -2.578299, -0.760540, 1.570796, 1.710782],accel_mss,speed_ms,0,blend_radius_m)
    movel([0.139757, -1.373922, -2.578040, -0.760426, 1.570796, 1.710554],accel_mss,speed_ms,0,blend_radius_m)
    movel([0.139564, -1.374300, -2.577777, -0.760312, 1.570796, 1.710361],accel_mss,speed_ms,0,blend_radius_m)
    movel([0.139410, -1.374677, -2.577515, -0.760197, 1.570796, 1.710206],accel_mss,speed_ms,0,blend_radius_m)
    movel([0.139295, -1.375052, -2.577254, -0.760084, 1.570796, 1.710091],accel_mss,speed_ms,0,blend_radius_m)
    movel([0.139220, -1.375414, -2.577001, -0.759974, 1.570796, 1.710017],accel_mss,speed_ms,0,blend_radius_m)
    movel([0.139188, -1.375768, -2.576754, -0.759867, 1.570796, 1.709984],accel_mss,speed_ms,0,blend_radius_m)
    movel([0.139200, -1.376104, -2.576519, -0.759766, 1.570796, 1.709996],accel_mss,speed_ms,0,blend_radius_m)
    movel([0.139250, -1.376425, -2.576295, -0.759669, 1.570796, 1.710046],accel_mss,speed_ms,0,blend_radius_m)
    movel([0.139348, -1.376733, -2.576079, -0.759577, 1.570796, 1.710144],accel_mss,speed_ms,0,blend_radius_m)
    movel([0.139488, -1.377016, -2.575881, -0.759492, 1.570796, 1.710284],accel_mss,speed_ms,0,blend_radius_m)
    movel([0.139673, -1.377273, -2.575701, -0.759415, 1.570796, 1.710469],accel_mss,speed_ms,0,blend_radius_m)
    movel([0.139898, -1.377502, -2.575540, -0.759346, 1.570796, 1.710695],accel_mss,speed_ms,0,blend_radius_m)
    movel([0.140160, -1.377700, -2.575402, -0.759287, 1.570796, 1.710956],accel_mss,speed_ms,0,blend_radius_m)
    movel([0.140456, -1.377861, -2.575289, -0.759239, 1.570796, 1.711252],accel_mss,speed_ms,0,blend_radius_m)
    movel([0.140782, -1.377988, -2.575200, -0.759201, 1.570796, 1.711578],accel_mss,speed_ms,0,blend_radius_m)
    movel([0.141137, -1.378076, -2.575138, -0.759175, 1.570796, 1.711934],accel_mss,speed_ms,0,blend_radius_m)
    movel([0.141514, -1.378124, -2.575104, -0.759160, 1.570796, 1.712310],accel_mss,speed_ms,0,blend_radius_m)
    movel([0.141920, -1.378136, -2.575096, -0.759157, 1.570796, 1.712716],accel_mss,speed_ms,0,blend_radius_m)
    movel([0.142340, -1.378109, -2.575115, -0.759165, 1.570796, 1.713136],accel_mss,speed_ms,0,blend_radius_m)
    movel([0.142773, -1.378045, -2.575160, -0.759184, 1.570796, 1.713569],accel_mss,speed_ms,0,blend_radius_m)
    movel([0.143214, -1.377943, -2.575231, -0.759214, 1.570796, 1.714011],accel_mss,speed_ms,0,blend_radius_m)
    movel([0.143660, -1.377804, -2.575329, -0.759256, 1.570796, 1.714456],accel_mss,speed_ms,0,blend_radius_m)
    movel([0.144106, -1.377629, -2.575451, -0.759308, 1.570796, 1.714903],accel_mss,speed_ms,0,blend_radius_m)
    movel([0.144549, -1.377422, -2.575597, -0.759370, 1.570796, 1.715345],accel_mss,speed_ms,0,blend_radius_m)
    movel([0.144987, -1.377181, -2.575765, -0.759442, 1.570796, 1.715783],accel_mss,speed_ms,0,blend_radius_m)
    movel([0.145417, -1.376907, -2.575957, -0.759525, 1.570796, 1.716213],accel_mss,speed_ms,0,blend_radius_m)
    movel([0.145830, -1.376607, -2.576167, -0.759615, 1.570796, 1.716626],accel_mss,speed_ms,0,blend_radius_m)
    movel([0.146222, -1.376282, -2.576394, -0.759712, 1.570796, 1.717019],accel_mss,speed_ms,0,blend_radius_m)
    movel([0.146587, -1.375941, -2.576633, -0.759815, 1.570796, 1.717383],accel_mss,speed_ms,0,blend_radius_m)
    movel([0.146918, -1.375586, -2.576880, -0.759922, 1.570796, 1.717715],accel_mss,speed_ms,0,blend_radius_m)
    movel([0.147221, -1.375215, -2.577139, -0.760034, 1.570796, 1.718017],accel_mss,speed_ms,0,blend_radius_m)
    movel([0.147490, -1.374833, -2.577406, -0.760150, 1.570796, 1.718286],accel_mss,speed_ms,0,blend_radius_m)
    movel([0.147725, -1.374436, -2.577683, -0.760270, 1.570796, 1.718521],accel_mss,speed_ms,0,blend_radius_m)
    movel([0.147922, -1.374037, -2.577961, -0.760392, 1.570796, 1.718719],accel_mss,speed_ms,0,blend_radius_m)
    movel([0.148071, -1.373653, -2.578227, -0.760508, 1.570796, 1.718868],accel_mss,speed_ms,0,blend_radius_m)
    movel([0.148177, -1.373272, -2.578493, -0.760625, 1.570796, 1.718973],accel_mss,speed_ms,0,blend_radius_m)
    movel([0.148237, -1.372899, -2.578752, -0.760739, 1.570796, 1.719033],accel_mss,speed_ms,0,blend_radius_m)
    movel([0.148252, -1.372539, -2.579001, -0.760849, 1.570796, 1.719048],accel_mss,speed_ms,0,blend_radius_m)
    movel([0.148218, -1.372197, -2.579238, -0.760953, 1.570796, 1.719014],accel_mss,speed_ms,0,blend_radius_m)
    movel([0.148139, -1.371877, -2.579460, -0.761052, 1.570796, 1.718936],accel_mss,speed_ms,0,blend_radius_m)
    movel([0.148139, -1.339270, -2.563771, -0.809348, 1.570796, 1.718936],accel_mss,speed_ms,0,blend_radius_m)
    speed_ms = 1.000
    movel([0.145797, -1.340501, -2.562957, -0.808931, 1.570796, 1.716594],accel_mss,speed_ms,0,blend_radius_m)
    speed_ms = 0.008
    movel([0.145797, -1.366938, -2.575821, -0.769630, 1.570796, 1.716594],accel_mss,speed_ms,0,blend_radius_m)
    speed_ms = 0.003
    movel([0.145797, -1.370274, -2.577353, -0.764762, 1.570796, 1.716594],accel_mss,speed_ms,0,blend_radius_m)
    speed_ms = 0.008
    movel([0.145665, -1.370067, -2.577496, -0.764826, 1.570796, 1.716462],accel_mss,speed_ms,0,blend_radius_m)
    movel([0.145416, -1.369838, -2.577654, -0.764897, 1.570796, 1.716212],accel_mss,speed_ms,0,blend_radius_m)
    movel([0.145110, -1.369642, -2.577790, -0.764957, 1.570796, 1.715907],accel_mss,speed_ms,0,blend_radius_m)
    movel([0.144825, -1.369529, -2.577868, -0.764992, 1.570796, 1.715621],accel_mss,speed_ms,0,blend_radius_m)
    movel([0.144417, -1.369437, -2.577931, -0.765021, 1.570796, 1.715214],accel_mss,speed_ms,0,blend_radius_m)
    movel([0.144164, -1.369418, -2.577944, -0.765026, 1.570796, 1.714961],accel_mss,speed_ms,0,blend_radius_m)
    movel([0.143888, -1.369480, -2.577901, -0.765007, 1.570796, 1.714685],accel_mss,speed_ms,0,blend_radius_m)
    movel([0.143604, -1.369621, -2.577804, -0.764964, 1.570796, 1.714401],accel_mss,speed_ms,0,blend_radius_m)
    movel([0.143314, -1.369805, -2.577677, -0.764907, 1.570796, 1.714110],accel_mss,speed_ms,0,blend_radius_m)
    movel([0.143042, -1.369990, -2.577550, -0.764850, 1.570796, 1.713838],accel_mss,speed_ms,0,blend_radius_m)
    movel([0.142613, -1.370337, -2.577309, -0.764742, 1.570796, 1.713410],accel_mss,speed_ms,0,blend_radius_m)
    movel([0.142405, -1.370539, -2.577170, -0.764680, 1.570796, 1.713201],accel_mss,speed_ms,0,blend_radius_m)
    movel([0.142211, -1.370751, -2.577023, -0.764615, 1.570796, 1.713007],accel_mss,speed_ms,0,blend_radius_m)
    movel([0.142030, -1.370976, -2.576867, -0.764546, 1.570796, 1.712826],accel_mss,speed_ms,0,blend_radius_m)
    movel([0.141750, -1.371410, -2.576567, -0.764413, 1.570796, 1.712546],accel_mss,speed_ms,0,blend_radius_m)
    movel([0.141560, -1.371856, -2.576257, -0.764276, 1.570796, 1.712356],accel_mss,speed_ms,0,blend_radius_m)
    movel([0.141472, -1.372280, -2.575963, -0.764146, 1.570796, 1.712268],accel_mss,speed_ms,0,blend_radius_m)
    movel([0.141491, -1.372656, -2.575702, -0.764031, 1.570796, 1.712287],accel_mss,speed_ms,0,blend_radius_m)
    movel([0.141607, -1.372963, -2.575488, -0.763938, 1.570796, 1.712404],accel_mss,speed_ms,0,blend_radius_m)
    movel([0.141800, -1.373198, -2.575325, -0.763866, 1.570796, 1.712597],accel_mss,speed_ms,0,blend_radius_m)
    movel([0.142061, -1.373372, -2.575204, -0.763813, 1.570796, 1.712858],accel_mss,speed_ms,0,blend_radius_m)
    movel([0.142382, -1.373473, -2.575133, -0.763783, 1.570796, 1.713178],accel_mss,speed_ms,0,blend_radius_m)
    movel([0.142758, -1.373499, -2.575115, -0.763775, 1.570796, 1.713554],accel_mss,speed_ms,0,blend_radius_m)
    movel([0.143174, -1.373452, -2.575148, -0.763789, 1.570796, 1.713971],accel_mss,speed_ms,0,blend_radius_m)
    movel([0.143605, -1.373330, -2.575233, -0.763826, 1.570796, 1.714402],accel_mss,speed_ms,0,blend_radius_m)
    movel([0.144041, -1.373140, -2.575365, -0.763884, 1.570796, 1.714837],accel_mss,speed_ms,0,blend_radius_m)
    movel([0.144465, -1.372885, -2.575543, -0.763962, 1.570796, 1.715261],accel_mss,speed_ms,0,blend_radius_m)
    movel([0.144862, -1.372577, -2.575757, -0.764056, 1.570796, 1.715659],accel_mss,speed_ms,0,blend_radius_m)
    movel([0.145208, -1.372234, -2.575995, -0.764160, 1.570796, 1.716004],accel_mss,speed_ms,0,blend_radius_m)
    movel([0.145490, -1.371866, -2.576250, -0.764273, 1.570796, 1.716287],accel_mss,speed_ms,0,blend_radius_m)
    movel([0.145708, -1.371480, -2.576518, -0.764391, 1.570796, 1.716505],accel_mss,speed_ms,0,blend_radius_m)
    movel([0.145843, -1.371102, -2.576780, -0.764507, 1.570796, 1.716640],accel_mss,speed_ms,0,blend_radius_m)
    movel([0.145893, -1.370746, -2.577026, -0.764617, 1.570796, 1.716689],accel_mss,speed_ms,0,blend_radius_m)
    movel([0.145853, -1.370418, -2.577253, -0.764718, 1.570796, 1.716649],accel_mss,speed_ms,0,blend_radius_m)
    movel([0.145797, -1.373079, -2.578626, -0.760683, 1.570796, 1.716594],accel_mss,speed_ms,0,blend_radius_m)
    movel([0.145665, -1.372873, -2.578769, -0.760746, 1.570796, 1.716462],accel_mss,speed_ms,0,blend_radius_m)
    movel([0.145416, -1.372644, -2.578928, -0.760816, 1.570796, 1.716212],accel_mss,speed_ms,0,blend_radius_m)
    movel([0.145110, -1.372449, -2.579064, -0.760876, 1.570796, 1.715907],accel_mss,speed_ms,0,blend_radius_m)
    movel([0.144825, -1.372336, -2.579142, -0.760911, 1.570796, 1.715621],accel_mss,speed_ms,0,blend_radius_m)
    movel([0.144417, -1.372244, -2.579206, -0.760939, 1.570796, 1.715214],accel_mss,speed_ms,0,blend_radius_m)
    movel([0.144164, -1.372226, -2.579218, -0.760945, 1.570796, 1.714961],accel_mss,speed_ms,0,blend_radius_m)
    movel([0.143888, -1.372288, -2.579176, -0.760926, 1.570796, 1.714685],accel_mss,speed_ms,0,blend_radius_m)
    movel([0.143604, -1.372428, -2.579078, -0.760883, 1.570796, 1.714401],accel_mss,speed_ms,0,blend_radius_m)
    movel([0.143314, -1.372611, -2.578951, -0.760827, 1.570796, 1.714110],accel_mss,speed_ms,0,blend_radius_m)
    movel([0.143042, -1.372796, -2.578823, -0.760770, 1.570796, 1.713838],accel_mss,speed_ms,0,blend_radius_m)
    movel([0.142613, -1.373143, -2.578582, -0.760664, 1.570796, 1.713410],accel_mss,speed_ms,0,blend_radius_m)
    movel([0.142405, -1.373344, -2.578443, -0.760603, 1.570796, 1.713201],accel_mss,speed_ms,0,blend_radius_m)
    movel([0.142211, -1.373556, -2.578295, -0.760538, 1.570796, 1.713007],accel_mss,speed_ms,0,blend_radius_m)
    movel([0.142030, -1.373779, -2.578140, -0.760470, 1.570796, 1.712826],accel_mss,speed_ms,0,blend_radius_m)
    movel([0.141750, -1.374213, -2.577838, -0.760338, 1.570796, 1.712546],accel_mss,speed_ms,0,blend_radius_m)
    movel([0.141560, -1.374657, -2.577528, -0.760203, 1.570796, 1.712356],accel_mss,speed_ms,0,blend_radius_m)
    movel([0.141472, -1.375081, -2.577233, -0.760075, 1.570796, 1.712268],accel_mss,speed_ms,0,blend_radius_m)
    movel([0.141491, -1.375456, -2.576971, -0.759961, 1.570796, 1.712287],accel_mss,speed_ms,0,blend_radius_m)
    movel([0.141607, -1.375763, -2.576757, -0.759869, 1.570796, 1.712404],accel_mss,speed_ms,0,blend_radius_m)
    movel([0.141800, -1.375997, -2.576594, -0.759798, 1.570796, 1.712597],accel_mss,speed_ms,0,blend_radius_m)
    movel([0.142061, -1.376170, -2.576473, -0.759746, 1.570796, 1.712858],accel_mss,speed_ms,0,blend_radius_m)
    movel([0.142382, -1.376271, -2.576402, -0.759716, 1.570796, 1.713178],accel_mss,speed_ms,0,blend_radius_m)
    movel([0.142758, -1.376297, -2.576384, -0.759708, 1.570796, 1.713554],accel_mss,speed_ms,0,blend_radius_m)
    movel([0.143174, -1.376250, -2.576417, -0.759722, 1.570796, 1.713971],accel_mss,speed_ms,0,blend_radius_m)
    movel([0.143605, -1.376129, -2.576502, -0.759758, 1.570796, 1.714402],accel_mss,speed_ms,0,blend_radius_m)
    movel([0.144041, -1.375939, -2.576634, -0.759816, 1.570796, 1.714837],accel_mss,speed_ms,0,blend_radius_m)
    movel([0.144465, -1.375684, -2.576812, -0.759892, 1.570796, 1.715261],accel_mss,speed_ms,0,blend_radius_m)
    movel([0.144862, -1.375377, -2.577027, -0.759985, 1.570796, 1.715659],accel_mss,speed_ms,0,blend_radius_m)
    movel([0.145208, -1.375035, -2.577265, -0.760089, 1.570796, 1.716004],accel_mss,speed_ms,0,blend_radius_m)
    movel([0.145490, -1.374668, -2.577521, -0.760200, 1.570796, 1.716287],accel_mss,speed_ms,0,blend_radius_m)
    movel([0.145708, -1.374283, -2.577789, -0.760317, 1.570796, 1.716505],accel_mss,speed_ms,0,blend_radius_m)
    movel([0.145843, -1.373905, -2.578052, -0.760432, 1.570796, 1.716640],accel_mss,speed_ms,0,blend_radius_m)
    movel([0.145893, -1.373550, -2.578299, -0.760540, 1.570796, 1.716689],accel_mss,speed_ms,0,blend_radius_m)
    movel([0.145853, -1.373223, -2.578526, -0.760639, 1.570796, 1.716649],accel_mss,speed_ms,0,blend_radius_m)
    movel([0.145797, -1.340501, -2.562957, -0.808931, 1.570796, 1.716594],accel_mss,speed_ms,0,blend_radius_m)
    speed_ms = 1.000
    movel([0.146700, -1.341961, -2.561990, -0.808439, 1.570796, 1.717496],accel_mss,speed_ms,0,blend_radius_m)
    speed_ms = 0.008
    movel([0.146700, -1.368370, -2.574834, -0.769184, 1.570796, 1.717496],accel_mss,speed_ms,0,blend_radius_m)
    speed_ms = 0.003
    movel([0.146700, -1.371702, -2.576364, -0.764323, 1.570796, 1.717496],accel_mss,speed_ms,0,blend_radius_m)
    speed_ms = 0.008
    movel([0.146515, -1.372001, -2.576156, -0.764231, 1.570796, 1.717312],accel_mss,speed_ms,0,blend_radius_m)
    movel([0.146310, -1.372296, -2.575951, -0.764141, 1.570796, 1.717106],accel_mss,speed_ms,0,blend_radius_m)
    movel([0.146072, -1.372595, -2.575744, -0.764050, 1.570796, 1.716868],accel_mss,speed_ms,0,blend_radius_m)
    movel([0.145854, -1.372836, -2.575577, -0.763976, 1.570796, 1.716651],accel_mss,speed_ms,0,blend_radius_m)
    movel([0.145623, -1.373056, -2.575423, -0.763909, 1.570796, 1.716419],accel_mss,speed_ms,0,blend_radius_m)
    movel([0.145375, -1.373262, -2.575281, -0.763847, 1.570796, 1.716171],accel_mss,speed_ms,0,blend_radius_m)
    movel([0.145105, -1.373453, -2.575147, -0.763789, 1.570796, 1.715901],accel_mss,speed_ms,0,blend_radius_m)
    movel([0.144824, -1.373626, -2.575027, -0.763736, 1.570796, 1.715620],accel_mss,speed_ms,0,blend_radius_m)
    movel([0.144503, -1.373792, -2.574911, -0.763686, 1.570796, 1.715300],accel_mss,speed_ms,0,blend_radius_m)
    movel([0.144154, -1.373941, -2.574807, -0.763640, 1.570796, 1.714951],accel_mss,speed_ms,0,blend_radius_m)
    movel([0.143741, -1.374090, -2.574704, -0.763595, 1.570796, 1.714537],accel_mss,speed_ms,0,blend_radius_m)
    movel([0.143329, -1.374212, -2.574618, -0.763558, 1.570796, 1.714125],accel_mss,speed_ms,0,blend_radius_m)
    movel([0.142981, -1.374296, -2.574560, -0.763533, 1.570796, 1.713778],accel_mss,speed_ms,0,blend_radius_m)
    movel([0.142643, -1.374352, -2.574521, -0.763516, 1.570796, 1.713439],accel_mss,speed_ms,0,blend_radius_m)
    movel([0.142311, -1.374380, -2.574501, -0.763507, 1.570796, 1.713108],accel_mss,speed_ms,0,blend_radius_m)
    movel([0.141991, -1.374383, -2.574499, -0.763507, 1.570796, 1.712788],accel_mss,speed_ms,0,blend_radius_m)
    movel([0.141699, -1.374362, -2.574514, -0.763513, 1.570796, 1.712495],accel_mss,speed_ms,0,blend_radius_m)
    movel([0.141435, -1.374317, -2.574545, -0.763527, 1.570796, 1.712231],accel_mss,speed_ms,0,blend_radius_m)
    movel([0.141198, -1.374248, -2.574593, -0.763547, 1.570796, 1.711994],accel_mss,speed_ms,0,blend_radius_m)
    movel([0.140980, -1.374154, -2.574659, -0.763576, 1.570796, 1.711776],accel_mss,speed_ms,0,blend_radius_m)
    movel([0.140781, -1.374031, -2.574745, -0.763613, 1.570796, 1.711577],accel_mss,speed_ms,0,blend_radius_m)
    movel([0.140605, -1.373884, -2.574847, -0.763658, 1.570796, 1.711401],accel_mss,speed_ms,0,blend_radius_m)
    movel([0.140456, -1.373715, -2.574965, -0.763709, 1.570796, 1.711253],accel_mss,speed_ms,0,blend_radius_m)
    movel([0.140339, -1.373529, -2.575094, -0.763765, 1.570796, 1.711135],accel_mss,speed_ms,0,blend_radius_m)
    movel([0.140254, -1.373325, -2.575236, -0.763827, 1.570796, 1.711050],accel_mss,speed_ms,0,blend_radius_m)
    movel([0.140198, -1.373103, -2.575391, -0.763895, 1.570796, 1.710994],accel_mss,speed_ms,0,blend_radius_m)
    movel([0.140172, -1.372869, -2.575553, -0.763966, 1.570796, 1.710969],accel_mss,speed_ms,0,blend_radius_m)
    movel([0.140176, -1.372622, -2.575725, -0.764042, 1.570796, 1.710972],accel_mss,speed_ms,0,blend_radius_m)
    movel([0.140213, -1.372344, -2.575918, -0.764126, 1.570796, 1.711009],accel_mss,speed_ms,0,blend_radius_m)
    movel([0.140277, -1.372065, -2.576112, -0.764212, 1.570796, 1.711073],accel_mss,speed_ms,0,blend_radius_m)
    movel([0.140374, -1.371776, -2.576312, -0.764300, 1.570796, 1.711170],accel_mss,speed_ms,0,blend_radius_m)
